LIN {X 0,Y 185.969,Z 314.942,A -85,B 0,C 180,E1 -22131.302,E2 -22131.302} C_VEL
LIN {X 0,Y 186.152,Z 314.876,A -85,B 0,C 180,E1 -22137.833,E2 -22137.833} C_VEL
LIN {X 0,Y 186.371,Z 314.881,A -85,B 0,C 180,E1 -22139.996,E2 -22139.996} C_VEL
LIN {X 0,Y 185.873,Z 314.921,A -85,B 0,C 180,E1 -22144.333,E2 -22144.333} C_VEL
LIN {X 0,Y 185.96,Z 314.906,A -85,B 0,C 180,E1 -22148.691,E2 -22148.691} C_VEL
LIN {X 0,Y 185.713,Z 314.968,A -85,B 0,C 180,E1 -22153.12,E2 -22153.12} C_VEL
LIN {X 0,Y 185.648,Z 314.931,A -85,B 0,C 180,E1 -22157.625,E2 -22157.625} C_VEL
LIN {X 0,Y 185.544,Z 314.997,A -85,B 0,C 180,E1 -22162.254,E2 -22162.254} C_VEL
LIN {X 0,Y 185.482,Z 314.953,A -85,B 0,C 180,E1 -22167.04,E2 -22167.04} C_VEL
LIN {X 0,Y 185.522,Z 315.001,A -85,B 0,C 180,E1 -22172.024,E2 -22172.024} C_VEL
LIN {X 0,Y 185.491,Z 314.96,A -85,B 0,C 180,E1 -22177.311,E2 -22177.311} C_VEL
LIN {X 0,Y 185.452,Z 315.01,A -85,B 0,C 180,E1 -22180.718,E2 -22180.718} C_VEL
LIN {X 0,Y 185.446,Z 314.975,A -85,B 0,C 180,E1 -22186.053,E2 -22186.053} C_VEL
LIN {X 0,Y 185.455,Z 315.011,A -85,B 0,C 180,E1 -22189.892,E2 -22189.892} C_VEL
LIN {X 0,Y 185.509,Z 315.032,A -85,B 0,C 180,E1 -22194.939,E2 -22194.939} C_VEL
LIN {X 0,Y 186.259,Z 317.419,A -85,B 0,C 180,E1 -22195.462,E2 -22195.462} C_VEL
LIN {X 0,Y 188.139,Z 319.677,A -85,B 0,C 180,E1 -22196.456,E2 -22196.456} C_VEL
LIN {X 0,Y 189.457,Z 320.605,A -85,B 0,C 180,E1 -22197.082,E2 -22197.082} C_VEL
LIN {X 0,Y 191.419,Z 323.893,A -85,B 0,C 180,E1 -22198.11,E2 -22198.11} C_VEL
LIN {X 0,Y 193.286,Z 325.807,A -85,B 0,C 180,E1 -22198.984,E2 -22198.984} C_VEL
LIN {X 0,Y 195.811,Z 329.375,A -85,B 0,C 180,E1 -22200.184,E2 -22200.184} C_VEL
LIN {X 0,Y 197.081,Z 331.066,A -85,B 0,C 180,E1 -22200.76,E2 -22200.76} C_VEL
LIN {X 0,Y 203.014,Z 339.247,A -85,B 0,C 180,E1 -22203.293,E2 -22203.293} C_VEL
LIN {X 0,Y 211.718,Z 352.303,A -85,B 0,C 180,E1 -22206.675,E2 -22206.675} C_VEL
LIN {X 0,Y 219.05,Z 364.426,A -85,B 0,C 180,E1 -22209.272,E2 -22209.272} C_VEL
LIN {X 0,Y 227.054,Z 378.808,A -85,B 0,C 180,E1 -22211.875,E2 -22211.875} C_VEL
LIN {X 0,Y 229.793,Z 385.325,A -85,B 0,C 180,E1 -22212.786,E2 -22212.786} C_VEL
LIN {X 0,Y 224.005,Z 468.269,A -85,B 0,C 180,E1 -22215.304,E2 -22215.304} C_VEL
LIN {X 0,Y 222.037,Z 484.164,A -85,B 0,C 180,E1 -22216.092,E2 -22216.092} C_VEL
LIN {X 0,Y 219.583,Z 498.974,A -85,B 0,C 180,E1 -22217.171,E2 -22217.171} C_VEL
LIN {X 0,Y 216.53,Z 513.139,A -85,B 0,C 180,E1 -22218.533,E2 -22218.533} C_VEL
LIN {X 0,Y 213.108,Z 526.59,A -85,B 0,C 180,E1 -22220.206,E2 -22220.206} C_VEL
LIN {X 0,Y 209.135,Z 539.856,A -85,B 0,C 180,E1 -22222.274,E2 -22222.274} C_VEL
LIN {X 0,Y 204.964,Z 552.181,A -85,B 0,C 180,E1 -22224.68,E2 -22224.68} C_VEL
LIN {X 0,Y 200.711,Z 563.728,A -85,B 0,C 180,E1 -22227.491,E2 -22227.491} C_VEL
LIN {X 0,Y 196.778,Z 573.885,A -85,B 0,C 180,E1 -22230.568,E2 -22230.568} C_VEL
LIN {X 0,Y 192.849,Z 583.499,A -85,B 0,C 180,E1 -22234.179,E2 -22234.179} C_VEL
LIN {X 0,Y 189.543,Z 591.563,A -85,B 0,C 180,E1 -22237.992,E2 -22237.992} C_VEL
LIN {X 0,Y 186.875,Z 598.44,A -85,B 0,C 180,E1 -22242.115,E2 -22242.115} C_VEL
LIN {X 0,Y 184.929,Z 604.134,A -85,B 0,C 180,E1 -22246.559,E2 -22246.559} C_VEL
LIN {X 0,Y 183.833,Z 607.594,A -85,B 0,C 180,E1 -22250.124,E2 -22250.124} C_VEL
LIN {X 0,Y 183.14,Z 609.731,A -85,B 0,C 180,E1 -22252.939,E2 -22252.939} C_VEL
LIN {X 0,Y 182.593,Z 612.209,A -85,B 0,C 180,E1 -22257.725,E2 -22257.725} C_VEL
LIN {X 0,Y 182.636,Z 613.322,A -85,B 0,C 180,E1 -22262.595,E2 -22262.595} C_VEL
LIN {X 0,Y 183.097,Z 613.279,A -85,B 0,C 180,E1 -22266.295,E2 -22266.295} C_VEL
LIN {X 0,Y 184.09,Z 612.207,A -85,B 0,C 180,E1 -22270.465,E2 -22270.465} C_VEL
LIN {X 0,Y 185.447,Z 610.546,A -85,B 0,C 180,E1 -22273.947,E2 -22273.947} C_VEL
LIN {X 0,Y 187.89,Z 607.254,A -85,B 0,C 180,E1 -22278.423,E2 -22278.423} C_VEL
LIN {X 0,Y 190.855,Z 603.121,A -85,B 0,C 180,E1 -22282.343,E2 -22282.343} C_VEL
LIN {X 0,Y 195.336,Z 596.767,A -85,B 0,C 180,E1 -22286.819,E2 -22286.819} C_VEL
LIN {X 0,Y 200.792,Z 588.688,A -85,B 0,C 180,E1 -22291.045,E2 -22291.045} C_VEL
LIN {X 0,Y 206.353,Z 580.032,A -85,B 0,C 180,E1 -22294.488,E2 -22294.488} C_VEL
LIN {X 0,Y 211.756,Z 570.942,A -85,B 0,C 180,E1 -22297.349,E2 -22297.349} C_VEL
LIN {X 0,Y 217.718,Z 560.022,A -85,B 0,C 180,E1 -22300.073,E2 -22300.073} C_VEL
LIN {X 0,Y 223.783,Z 547.561,A -85,B 0,C 180,E1 -22302.536,E2 -22302.536} C_VEL
LIN {X 0,Y 229.323,Z 534.602,A -85,B 0,C 180,E1 -22304.538,E2 -22304.538} C_VEL
LIN {X 0,Y 234.001,Z 521.869,A -85,B 0,C 180,E1 -22306.101,E2 -22306.101} C_VEL
LIN {X 0,Y 238.248,Z 507.978,A -85,B 0,C 180,E1 -22307.443,E2 -22307.443} C_VEL
LIN {X 0,Y 241.757,Z 493.694,A -85,B 0,C 180,E1 -22308.498,E2 -22308.498} C_VEL
LIN {X 0,Y 244.702,Z 478.011,A -85,B 0,C 180,E1 -22309.327,E2 -22309.327} C_VEL
LIN {X 0,Y 246.667,Z 461.81,A -85,B 0,C 180,E1 -22309.898,E2 -22309.898} C_VEL
LIN {X 0,Y 252.263,Z 398.759,A -85,B 0,C 180,E1 -22311.644,E2 -22311.644} C_VEL
LIN {X 0,Y 250.263,Z 393.549,A -85,B 0,C 180,E1 -22312.821,E2 -22312.821} C_VEL
LIN {X 0,Y 246.472,Z 386.354,A -85,B 0,C 180,E1 -22315.096,E2 -22315.096} C_VEL
LIN {X 0,Y 242.393,Z 379.192,A -85,B 0,C 180,E1 -22317.911,E2 -22317.911} C_VEL
LIN {X 0,Y 240.443,Z 376.102,A -85,B 0,C 180,E1 -22319.444,E2 -22319.444} C_VEL
LIN {X 0,Y 237.536,Z 371.34,A -85,B 0,C 180,E1 -22322.141,E2 -22322.141} C_VEL
LIN {X 0,Y 235.778,Z 368.411,A -85,B 0,C 180,E1 -22324.111,E2 -22324.111} C_VEL
LIN {X 0,Y 233.394,Z 365.664,A -85,B 0,C 180,E1 -22327.468,E2 -22327.468} C_VEL
LIN {X 0,Y 232.588,Z 363.6,A -85,B 0,C 180,E1 -22329.388,E2 -22329.388} C_VEL
LIN {X 0,Y 231.393,Z 363.089,A -85,B 0,C 180,E1 -22335.867,E2 -22335.867} C_VEL
LIN {X 0,Y 232.583,Z 363.999,A -85,B 0,C 180,E1 -22340.339,E2 -22340.339} C_VEL
LIN {X 0,Y 234.637,Z 367.807,A -85,B 0,C 180,E1 -22344.159,E2 -22344.159} C_VEL
LIN {X 0,Y 236.244,Z 370.311,A -85,B 0,C 180,E1 -22346.214,E2 -22346.214} C_VEL
LIN {X 0,Y 239.041,Z 375.498,A -85,B 0,C 180,E1 -22349.15,E2 -22349.15} C_VEL
LIN {X 0,Y 241.266,Z 379.857,A -85,B 0,C 180,E1 -22351.073,E2 -22351.073} C_VEL
LIN {X 0,Y 244.66,Z 386.769,A -85,B 0,C 180,E1 -22353.626,E2 -22353.626} C_VEL
LIN {X 0,Y 245.434,Z 389.581,A -85,B 0,C 180,E1 -22354.248,E2 -22354.248} C_VEL
LIN {X 0,Y 246.014,Z 395.44,A -85,B 0,C 180,E1 -22354.985,E2 -22354.985} C_VEL
LIN {X 0,Y 246.682,Z 402.682,A -85,B 0,C 180,E1 -22355.839,E2 -22355.839} C_VEL
LIN {X 0,Y 247.202,Z 404.751,A -85,B 0,C 180,E1 -22356.22,E2 -22356.22} C_VEL
LIN {X 0,Y 248.199,Z 407.486,A -85,B 0,C 180,E1 -22356.843,E2 -22356.843} C_VEL
LIN {X 0,Y 241.718,Z 476.664,A -85,B 0,C 180,E1 -22358.781,E2 -22358.781} C_VEL
LIN {X 0,Y 239.106,Z 492.462,A -85,B 0,C 180,E1 -22359.425,E2 -22359.425} C_VEL
LIN {X 0,Y 235.556,Z 507.607,A -85,B 0,C 180,E1 -22360.302,E2 -22360.302} C_VEL
LIN {X 0,Y 230.993,Z 522.645,A -85,B 0,C 180,E1 -22361.48,E2 -22361.48} C_VEL
LIN {X 0,Y 226.376,Z 535.543,A -85,B 0,C 180,E1 -22362.826,E2 -22362.826} C_VEL
LIN {X 0,Y 220.654,Z 549.173,A -85,B 0,C 180,E1 -22364.649,E2 -22364.649} C_VEL
LIN {X 0,Y 214.991,Z 560.943,A -85,B 0,C 180,E1 -22366.65,E2 -22366.65} C_VEL
LIN {X 0,Y 209.039,Z 572.068,A -85,B 0,C 180,E1 -22369.037,E2 -22369.037} C_VEL
LIN {X 0,Y 203.445,Z 581.51,A -85,B 0,C 180,E1 -22371.554,E2 -22371.554} C_VEL
LIN {X 0,Y 197.508,Z 590.878,A -85,B 0,C 180,E1 -22374.676,E2 -22374.676} C_VEL
LIN {X 0,Y 193.038,Z 597.736,A -85,B 0,C 180,E1 -22377.522,E2 -22377.522} C_VEL
LIN {X 0,Y 188.313,Z 604.455,A -85,B 0,C 180,E1 -22380.978,E2 -22380.978} C_VEL
LIN {X 0,Y 183.914,Z 610.718,A -85,B 0,C 180,E1 -22385.145,E2 -22385.145} C_VEL
LIN {X 0,Y 180.456,Z 615.636,A -85,B 0,C 180,E1 -22389.483,E2 -22389.483} C_VEL
LIN {X 0,Y 178.06,Z 619.319,A -85,B 0,C 180,E1 -22393.962,E2 -22393.962} C_VEL
LIN {X 0,Y 176.576,Z 621.83,A -85,B 0,C 180,E1 -22398.522,E2 -22398.522} C_VEL
LIN {X 0,Y 175.946,Z 623.194,A -85,B 0,C 180,E1 -22403.119,E2 -22403.119} C_VEL
LIN {X 0,Y 175.957,Z 623.379,A -85,B 0,C 180,E1 -22407.712,E2 -22407.712} C_VEL
LIN {X 0,Y 176.109,Z 623.043,A -85,B 0,C 180,E1 -22410.001,E2 -22410.001} C_VEL
LIN {X 0,Y 175.952,Z 621.46,A -85,B 0,C 180,E1 -22414.583,E2 -22414.583} C_VEL
LIN {X 0,Y 176.214,Z 618.649,A -85,B 0,C 180,E1 -22419.181,E2 -22419.181} C_VEL
LIN {X 0,Y 177.095,Z 614.534,A -85,B 0,C 180,E1 -22423.776,E2 -22423.776} C_VEL
LIN {X 0,Y 178.863,Z 609.007,A -85,B 0,C 180,E1 -22428.322,E2 -22428.322} C_VEL
LIN {X 0,Y 181.558,Z 601.914,A -85,B 0,C 180,E1 -22432.774,E2 -22432.774} C_VEL
LIN {X 0,Y 184.649,Z 594.281,A -85,B 0,C 180,E1 -22436.566,E2 -22436.566} C_VEL
LIN {X 0,Y 188.581,Z 585.073,A -85,B 0,C 180,E1 -22440.207,E2 -22440.207} C_VEL
LIN {X 0,Y 192.358,Z 575.617,A -85,B 0,C 180,E1 -22443.233,E2 -22443.233} C_VEL
LIN {X 0,Y 196.738,Z 564.464,A -85,B 0,C 180,E1 -22446.116,E2 -22446.116} C_VEL
LIN {X 0,Y 201.25,Z 552.272,A -85,B 0,C 180,E1 -22448.625,E2 -22448.625} C_VEL
LIN {X 0,Y 205.144,Z 540.321,A -85,B 0,C 180,E1 -22450.611,E2 -22450.611} C_VEL
LIN {X 0,Y 208.785,Z 527.578,A -85,B 0,C 180,E1 -22452.317,E2 -22452.317} C_VEL
LIN {X 0,Y 212.174,Z 513.906,A -85,B 0,C 180,E1 -22453.745,E2 -22453.745} C_VEL
LIN {X 0,Y 215.168,Z 499.638,A -85,B 0,C 180,E1 -22454.855,E2 -22454.855} C_VEL
LIN {X 0,Y 217.464,Z 484.324,A -85,B 0,C 180,E1 -22455.729,E2 -22455.729} C_VEL
LIN {X 0,Y 219.024,Z 466.927,A -85,B 0,C 180,E1 -22456.384,E2 -22456.384} C_VEL
LIN {X 0,Y 224.02,Z 395.336,A -85,B 0,C 180,E1 -22458.576,E2 -22458.576} C_VEL
LIN {X 0,Y 218.08,Z 380.998,A -85,B 0,C 180,E1 -22460.678,E2 -22460.678} C_VEL
LIN {X 0,Y 211.283,Z 366.529,A -85,B 0,C 180,E1 -22463.217,E2 -22463.217} C_VEL
LIN {X 0,Y 204.623,Z 353.731,A -85,B 0,C 180,E1 -22465.876,E2 -22465.876} C_VEL
LIN {X 0,Y 199.25,Z 344.249,A -85,B 0,C 180,E1 -22468.184,E2 -22468.184} C_VEL
LIN {X 0,Y 192.162,Z 334.537,A -85,B 0,C 180,E1 -22471.394,E2 -22471.394} C_VEL
LIN {X 0,Y 189.576,Z 330.921,A -85,B 0,C 180,E1 -22472.689,E2 -22472.689} C_VEL
LIN {X 0,Y 186.864,Z 327.443,A -85,B 0,C 180,E1 -22474.07,E2 -22474.07} C_VEL
LIN {X 0,Y 186.034,Z 326.335,A -85,B 0,C 180,E1 -22474.513,E2 -22474.513} C_VEL
LIN {X 0,Y 183.548,Z 323.572,A -85,B 0,C 180,E1 -22475.848,E2 -22475.848} C_VEL
LIN {X 0,Y 182.267,Z 321.267,A -85,B 0,C 180,E1 -22476.639,E2 -22476.639} C_VEL
LIN {X 0,Y 179.8,Z 319.198,A -85,B 0,C 180,E1 -22478.048,E2 -22478.048} C_VEL
LIN {X 0,Y 178.699,Z 317.03,A -85,B 0,C 180,E1 -22478.814,E2 -22478.814} C_VEL
LIN {X 0,Y 178.468,Z 315.883,A -85,B 0,C 180,E1 -22479.088,E2 -22479.088} C_VEL
LIN {X 0,Y 178.608,Z 315.862,A -85,B 0,C 180,E1 -22481.648,E2 -22481.648} C_VEL
LIN {X 0,Y 178.637,Z 315.809,A -85,B 0,C 180,E1 -22486.343,E2 -22486.343} C_VEL
LIN {X 0,Y 178.901,Z 315.815,A -85,B 0,C 180,E1 -22490.956,E2 -22490.956} C_VEL
LIN {X 0,Y 178.809,Z 315.792,A -85,B 0,C 180,E1 -22495.488,E2 -22495.488} C_VEL
LIN {X 0,Y 179.337,Z 315.755,A -85,B 0,C 180,E1 -22499.996,E2 -22499.996} C_VEL
LIN {X 0,Y 178.822,Z 315.795,A -85,B 0,C 180,E1 -22504.504,E2 -22504.504} C_VEL
LIN {X 0,Y 178.893,Z 315.79,A -85,B 0,C 180,E1 -22509.037,E2 -22509.037} C_VEL
LIN {X 0,Y 178.639,Z 315.838,A -85,B 0,C 180,E1 -22513.65,E2 -22513.65} C_VEL
LIN {X 0,Y 178.551,Z 315.829,A -85,B 0,C 180,E1 -22519.149,E2 -22519.149} C_VEL
LIN {X 0,Y 178.457,Z 315.841,A -85,B 0,C 180,E1 -22525.071,E2 -22525.071} C_VEL
LIN {X 0,Y 178.442,Z 315.872,A -85,B 0,C 180,E1 -22530.793,E2 -22530.793} C_VEL
LIN {X 0,Y 178.474,Z 315.852,A -85,B 0,C 180,E1 -22534.214,E2 -22534.214} C_VEL
LIN {X 0,Y 178.378,Z 315.863,A -85,B 0,C 180,E1 -22539.073,E2 -22539.073} C_VEL
LIN {X 0,Y 178.383,Z 315.887,A -85,B 0,C 180,E1 -22542.043,E2 -22542.043} C_VEL
LIN {X 0,Y 178.381,Z 315.853,A -85,B 0,C 180,E1 -22545.162,E2 -22545.162} C_VEL
LIN {X 0,Y 178.391,Z 315.884,A -85,B 0,C 180,E1 -22548.457,E2 -22548.457} C_VEL
LIN {X 0,Y 178.427,Z 316.051,A -85,B 0,C 180,E1 -22551.495,E2 -22551.495} C_VEL
LIN {X 0,Y 179.26,Z 318.459,A -85,B 0,C 180,E1 -22552.133,E2 -22552.133} C_VEL
LIN {X 0,Y 181.378,Z 320.729,A -85,B 0,C 180,E1 -22553.398,E2 -22553.398} C_VEL
LIN {X 0,Y 182.523,Z 321.562,A -85,B 0,C 180,E1 -22554.03,E2 -22554.03} C_VEL
LIN {X 0,Y 184.397,Z 324.755,A -85,B 0,C 180,E1 -22555.164,E2 -22555.164} C_VEL
LIN {X 0,Y 186.648,Z 327.025,A -85,B 0,C 180,E1 -22556.342,E2 -22556.342} C_VEL
LIN {X 0,Y 189.277,Z 330.678,A -85,B 0,C 180,E1 -22557.712,E2 -22557.712} C_VEL
LIN {X 0,Y 190.556,Z 332.255,A -85,B 0,C 180,E1 -22558.336,E2 -22558.336} C_VEL
LIN {X 0,Y 194.712,Z 338.031,A -85,B 0,C 180,E1 -22560.336,E2 -22560.336} C_VEL
LIN {X 0,Y 199.594,Z 344.846,A -85,B 0,C 180,E1 -22562.492,E2 -22562.492} C_VEL
LIN {X 0,Y 207.433,Z 356.74,A -85,B 0,C 180,E1 -22565.674,E2 -22565.674} C_VEL
LIN {X 0,Y 214.405,Z 368.342,A -85,B 0,C 180,E1 -22568.253,E2 -22568.253} C_VEL
LIN {X 0,Y 222.471,Z 383.07,A -85,B 0,C 180,E1 -22571.011,E2 -22571.011} C_VEL
LIN {X 0,Y 224.336,Z 387.564,A -85,B 0,C 180,E1 -22571.654,E2 -22571.654} C_VEL
LIN {X 0,Y 218.461,Z 468.888,A -85,B 0,C 180,E1 -22574.166,E2 -22574.166} C_VEL
LIN {X 0,Y 216.47,Z 484.361,A -85,B 0,C 180,E1 -22574.945,E2 -22574.945} C_VEL
LIN {X 0,Y 213.834,Z 499.73,A -85,B 0,C 180,E1 -22576.093,E2 -22576.093} C_VEL
LIN {X 0,Y 211.126,Z 511.825,A -85,B 0,C 180,E1 -22577.259,E2 -22577.259} C_VEL
LIN {X 0,Y 207.236,Z 526.822,A -85,B 0,C 180,E1 -22579.128,E2 -22579.128} C_VEL
LIN {X 0,Y 203.009,Z 540.396,A -85,B 0,C 180,E1 -22581.288,E2 -22581.288} C_VEL
LIN {X 0,Y 198.447,Z 553.329,A -85,B 0,C 180,E1 -22583.9,E2 -22583.9} C_VEL
LIN {X 0,Y 193.911,Z 565.051,A -85,B 0,C 180,E1 -22586.883,E2 -22586.883} C_VEL
LIN {X 0,Y 189.741,Z 575.331,A -85,B 0,C 180,E1 -22590.159,E2 -22590.159} C_VEL
LIN {X 0,Y 185.825,Z 584.495,A -85,B 0,C 180,E1 -22593.794,E2 -22593.794} C_VEL
LIN {X 0,Y 182.463,Z 592.427,A -85,B 0,C 180,E1 -22597.747,E2 -22597.747} C_VEL
LIN {X 0,Y 179.701,Z 599.325,A -85,B 0,C 180,E1 -22602.136,E2 -22602.136} C_VEL
LIN {X 0,Y 177.99,Z 604.089,A -85,B 0,C 180,E1 -22606.044,E2 -22606.044} C_VEL
LIN {X 0,Y 176.833,Z 607.616,A -85,B 0,C 180,E1 -22609.743,E2 -22609.743} C_VEL
LIN {X 0,Y 175.927,Z 610.358,A -85,B 0,C 180,E1 -22613.544,E2 -22613.544} C_VEL
LIN {X 0,Y 175.474,Z 612.543,A -85,B 0,C 180,E1 -22618.23,E2 -22618.23} C_VEL
LIN {X 0,Y 175.548,Z 613.516,A -85,B 0,C 180,E1 -22622.792,E2 -22622.792} C_VEL
LIN {X 0,Y 176.116,Z 613.448,A -85,B 0,C 180,E1 -22627.058,E2 -22627.058} C_VEL
LIN {X 0,Y 177.599,Z 611.991,A -85,B 0,C 180,E1 -22632.276,E2 -22632.276} C_VEL
LIN {X 0,Y 178.81,Z 610.595,A -85,B 0,C 180,E1 -22635.027,E2 -22635.027} C_VEL
LIN {X 0,Y 180.831,Z 608.066,A -85,B 0,C 180,E1 -22638.652,E2 -22638.652} C_VEL
LIN {X 0,Y 184.315,Z 603.615,A -85,B 0,C 180,E1 -22643.197,E2 -22643.197} C_VEL
LIN {X 0,Y 188.248,Z 598.396,A -85,B 0,C 180,E1 -22647.137,E2 -22647.137} C_VEL
LIN {X 0,Y 193.013,Z 591.885,A -85,B 0,C 180,E1 -22650.91,E2 -22650.91} C_VEL
LIN {X 0,Y 198.528,Z 583.958,A -85,B 0,C 180,E1 -22654.46,E2 -22654.46} C_VEL
LIN {X 0,Y 204.857,Z 574.171,A -85,B 0,C 180,E1 -22657.857,E2 -22657.857} C_VEL
LIN {X 0,Y 211.014,Z 563.701,A -85,B 0,C 180,E1 -22660.709,E2 -22660.709} C_VEL
LIN {X 0,Y 216.818,Z 552.838,A -85,B 0,C 180,E1 -22663.042,E2 -22663.042} C_VEL
LIN {X 0,Y 222.305,Z 541.16,A -85,B 0,C 180,E1 -22665.069,E2 -22665.069} C_VEL
LIN {X 0,Y 227.416,Z 528.817,A -85,B 0,C 180,E1 -22666.763,E2 -22666.763} C_VEL
LIN {X 0,Y 232.428,Z 514.442,A -85,B 0,C 180,E1 -22668.321,E2 -22668.321} C_VEL
LIN {X 0,Y 236.635,Z 499.469,A -85,B 0,C 180,E1 -22669.56,E2 -22669.56} C_VEL
LIN {X 0,Y 239.91,Z 484.566,A -85,B 0,C 180,E1 -22670.456,E2 -22670.456} C_VEL
LIN {X 0,Y 242.243,Z 469.817,A -85,B 0,C 180,E1 -22671.075,E2 -22671.075} C_VEL
LIN {X 0,Y 248.591,Z 401.712,A -85,B 0,C 180,E1 -22672.994,E2 -22672.994} C_VEL
LIN {X 0,Y 246.4,Z 396.681,A -85,B 0,C 180,E1 -22674.353,E2 -22674.353} C_VEL
LIN {X 0,Y 242.54,Z 389.311,A -85,B 0,C 180,E1 -22676.931,E2 -22676.931} C_VEL
LIN {X 0,Y 239.177,Z 383.222,A -85,B 0,C 180,E1 -22679.593,E2 -22679.593} C_VEL
LIN {X 0,Y 235.727,Z 377.515,A -85,B 0,C 180,E1 -22682.939,E2 -22682.939} C_VEL
LIN {X 0,Y 234.369,Z 375.198,A -85,B 0,C 180,E1 -22684.587,E2 -22684.587} C_VEL
LIN {X 0,Y 232.11,Z 372.295,A -85,B 0,C 180,E1 -22688.027,E2 -22688.027} C_VEL
LIN {X 0,Y 231.583,Z 370.675,A -85,B 0,C 180,E1 -22689.429,E2 -22689.429} C_VEL
LIN {X 0,Y 230.386,Z 370.078,A -85,B 0,C 180,E1 -22694.128,E2 -22694.128} C_VEL
LIN {X 0,Y 231.402,Z 370.743,A -85,B 0,C 180,E1 -22699.828,E2 -22699.828} C_VEL
LIN {X 0,Y 233.506,Z 374.763,A -85,B 0,C 180,E1 -22703.983,E2 -22703.983} C_VEL
LIN {X 0,Y 234.772,Z 377.041,A -85,B 0,C 180,E1 -22705.732,E2 -22705.732} C_VEL
LIN {X 0,Y 237.352,Z 381.993,A -85,B 0,C 180,E1 -22708.58,E2 -22708.58} C_VEL
LIN {X 0,Y 239.344,Z 386.127,A -85,B 0,C 180,E1 -22710.424,E2 -22710.424} C_VEL
LIN {X 0,Y 242.617,Z 393.253,A -85,B 0,C 180,E1 -22713.054,E2 -22713.054} C_VEL
LIN {X 0,Y 246.079,Z 401.676,A -85,B 0,C 180,E1 -22715.481,E2 -22715.481} C_VEL
LIN {X 0,Y 247.202,Z 404.751,A -85,B 0,C 180,E1 -22716.22,E2 -22716.22} C_VEL
LIN {X 0,Y 247.478,Z 407.165,A -85,B 0,C 180,E1 -22716.506,E2 -22716.506} C_VEL
LIN {X 0,Y 247.073,Z 410.629,A -85,B 0,C 180,E1 -22716.562,E2 -22716.562} C_VEL
LIN {X 0,Y 246.116,Z 414.43,A -85,B 0,C 180,E1 -22716.399,E2 -22716.399} C_VEL
LIN {X 0,Y 244.032,Z 421.322,A -85,B 0,C 180,E1 -22715.939,E2 -22715.939} C_VEL
LIN {X 0,Y 243.236,Z 425.628,A -85,B 0,C 180,E1 -22715.88,E2 -22715.88} C_VEL
LIN {X 0,Y 238.248,Z 476.462,A -85,B 0,C 180,E1 -22717.296,E2 -22717.296} C_VEL
LIN {X 0,Y 235.565,Z 492.245,A -85,B 0,C 180,E1 -22717.933,E2 -22717.933} C_VEL
LIN {X 0,Y 231.754,Z 507.931,A -85,B 0,C 180,E1 -22718.835,E2 -22718.835} C_VEL
LIN {X 0,Y 227.06,Z 522.856,A -85,B 0,C 180,E1 -22720.001,E2 -22720.001} C_VEL
LIN {X 0,Y 221.7,Z 537.042,A -85,B 0,C 180,E1 -22721.505,E2 -22721.505} C_VEL
LIN {X 0,Y 215.917,Z 550.055,A -85,B 0,C 180,E1 -22723.286,E2 -22723.286} C_VEL
LIN {X 0,Y 209.93,Z 561.87,A -85,B 0,C 180,E1 -22725.331,E2 -22725.331} C_VEL
LIN {X 0,Y 203.77,Z 572.85,A -85,B 0,C 180,E1 -22727.738,E2 -22727.738} C_VEL
LIN {X 0,Y 197.005,Z 583.594,A -85,B 0,C 180,E1 -22730.714,E2 -22730.714} C_VEL
LIN {X 0,Y 190.936,Z 592.566,A -85,B 0,C 180,E1 -22733.921,E2 -22733.921} C_VEL
LIN {X 0,Y 184.976,Z 601.064,A -85,B 0,C 180,E1 -22737.867,E2 -22737.867} C_VEL
LIN {X 0,Y 180.848,Z 606.356,A -85,B 0,C 180,E1 -22740.939,E2 -22740.939} C_VEL
LIN {X 0,Y 176.43,Z 612.193,A -85,B 0,C 180,E1 -22745.277,E2 -22745.277} C_VEL
LIN {X 0,Y 173.75,Z 615.698,A -85,B 0,C 180,E1 -22748.653,E2 -22748.653} C_VEL
LIN {X 0,Y 171.193,Z 619.285,A -85,B 0,C 180,E1 -22753.301,E2 -22753.301} C_VEL
LIN {X 0,Y 169.577,Z 621.717,A -85,B 0,C 180,E1 -22758.042,E2 -22758.042} C_VEL
LIN {X 0,Y 168.881,Z 623.027,A -85,B 0,C 180,E1 -22762.829,E2 -22762.829} C_VEL
LIN {X 0,Y 168.866,Z 623.155,A -85,B 0,C 180,E1 -22767.616,E2 -22767.616} C_VEL
LIN {X 0,Y 169.015,Z 622.782,A -85,B 0,C 180,E1 -22770.001,E2 -22770.001} C_VEL
LIN {X 0,Y 168.861,Z 621.126,A -85,B 0,C 180,E1 -22774.776,E2 -22774.776} C_VEL
LIN {X 0,Y 169.152,Z 618.239,A -85,B 0,C 180,E1 -22779.567,E2 -22779.567} C_VEL
LIN {X 0,Y 170.141,Z 614.043,A -85,B 0,C 180,E1 -22784.35,E2 -22784.35} C_VEL
LIN {X 0,Y 172.056,Z 608.427,A -85,B 0,C 180,E1 -22789.074,E2 -22789.074} C_VEL
LIN {X 0,Y 174.962,Z 601.239,A -85,B 0,C 180,E1 -22793.684,E2 -22793.684} C_VEL
LIN {X 0,Y 178.259,Z 593.51,A -85,B 0,C 180,E1 -22797.598,E2 -22797.598} C_VEL
LIN {X 0,Y 181.756,Z 585.608,A -85,B 0,C 180,E1 -22800.82,E2 -22800.82} C_VEL
LIN {X 0,Y 185.713,Z 576.159,A -85,B 0,C 180,E1 -22803.984,E2 -22803.984} C_VEL
LIN {X 0,Y 190.167,Z 565.306,A -85,B 0,C 180,E1 -22806.909,E2 -22806.909} C_VEL
LIN {X 0,Y 194.79,Z 553.313,A -85,B 0,C 180,E1 -22809.487,E2 -22809.487} C_VEL
LIN {X 0,Y 199.276,Z 540.18,A -85,B 0,C 180,E1 -22811.734,E2 -22811.734} C_VEL
LIN {X 0,Y 203.226,Z 526.764,A -85,B 0,C 180,E1 -22813.549,E2 -22813.549} C_VEL
LIN {X 0,Y 206.826,Z 512.678,A -85,B 0,C 180,E1 -22815.008,E2 -22815.008} C_VEL
LIN {X 0,Y 209.881,Z 498.053,A -85,B 0,C 180,E1 -22816.136,E2 -22816.136} C_VEL
LIN {X 0,Y 212.103,Z 483.191,A -85,B 0,C 180,E1 -22816.973,E2 -22816.973} C_VEL
LIN {X 0,Y 213.715,Z 465.346,A -85,B 0,C 180,E1 -22817.636,E2 -22817.636} C_VEL
LIN {X 0,Y 218.616,Z 397.485,A -85,B 0,C 180,E1 -22819.74,E2 -22819.74} C_VEL
LIN {X 0,Y 212.955,Z 383.809,A -85,B 0,C 180,E1 -22821.861,E2 -22821.861} C_VEL
LIN {X 0,Y 206.763,Z 370.469,A -85,B 0,C 180,E1 -22824.294,E2 -22824.294} C_VEL
LIN {X 0,Y 200.37,Z 357.844,A -85,B 0,C 180,E1 -22827.002,E2 -22827.002} C_VEL
LIN {X 0,Y 195.617,Z 349.465,A -85,B 0,C 180,E1 -22829.129,E2 -22829.129} C_VEL
LIN {X 0,Y 189.08,Z 340.322,A -85,B 0,C 180,E1 -22832.236,E2 -22832.236} C_VEL
LIN {X 0,Y 186.138,Z 336.31,A -85,B 0,C 180,E1 -22833.741,E2 -22833.741} C_VEL
LIN {X 0,Y 183.172,Z 332.349,A -85,B 0,C 180,E1 -22835.351,E2 -22835.351} C_VEL
LIN {X 0,Y 180.57,Z 329.169,A -85,B 0,C 180,E1 -22836.841,E2 -22836.841} C_VEL
LIN {X 0,Y 179.448,Z 327.418,A -85,B 0,C 180,E1 -22837.548,E2 -22837.548} C_VEL
LIN {X 0,Y 176.899,Z 324.763,A -85,B 0,C 180,E1 -22839.12,E2 -22839.12} C_VEL
LIN {X 0,Y 175.559,Z 322.336,A -85,B 0,C 180,E1 -22840.067,E2 -22840.067} C_VEL
LIN {X 0,Y 173.109,Z 320.353,A -85,B 0,C 180,E1 -22841.657,E2 -22841.657} C_VEL
LIN {X 0,Y 171.818,Z 318.022,A -85,B 0,C 180,E1 -22842.669,E2 -22842.669} C_VEL
LIN {X 0,Y 171.526,Z 316.748,A -85,B 0,C 180,E1 -22843.022,E2 -22843.022} C_VEL
LIN {X 0,Y 171.768,Z 316.67,A -85,B 0,C 180,E1 -22849.104,E2 -22849.104} C_VEL
LIN {X 0,Y 171.851,Z 316.699,A -85,B 0,C 180,E1 -22852.949,E2 -22852.949} C_VEL
LIN {X 0,Y 172.301,Z 316.629,A -85,B 0,C 180,E1 -22859.996,E2 -22859.996} C_VEL
LIN {X 0,Y 171.771,Z 316.669,A -85,B 0,C 180,E1 -22864.69,E2 -22864.69} C_VEL
LIN {X 0,Y 171.834,Z 316.674,A -85,B 0,C 180,E1 -22869.412,E2 -22869.412} C_VEL
LIN {X 0,Y 171.553,Z 316.707,A -85,B 0,C 180,E1 -22874.225,E2 -22874.225} C_VEL
LIN {X 0,Y 171.476,Z 316.714,A -85,B 0,C 180,E1 -22879.497,E2 -22879.497} C_VEL
LIN {X 0,Y 171.394,Z 316.714,A -85,B 0,C 180,E1 -22885.564,E2 -22885.564} C_VEL
LIN {X 0,Y 171.397,Z 316.744,A -85,B 0,C 180,E1 -22890.562,E2 -22890.562} C_VEL
LIN {X 0,Y 171.383,Z 316.723,A -85,B 0,C 180,E1 -22895.031,E2 -22895.031} C_VEL
LIN {X 0,Y 171.334,Z 316.734,A -85,B 0,C 180,E1 -22898.797,E2 -22898.797} C_VEL
LIN {X 0,Y 171.308,Z 316.737,A -85,B 0,C 180,E1 -22904.215,E2 -22904.215} C_VEL
LIN {X 0,Y 171.355,Z 316.886,A -85,B 0,C 180,E1 -22907.449,E2 -22907.449} C_VEL
LIN {X 0,Y 172.14,Z 319.223,A -85,B 0,C 180,E1 -22908.178,E2 -22908.178} C_VEL
LIN {X 0,Y 174.009,Z 321.478,A -85,B 0,C 180,E1 -22909.52,E2 -22909.52} C_VEL
LIN {X 0,Y 175.727,Z 322.713,A -85,B 0,C 180,E1 -22910.609,E2 -22910.609} C_VEL
LIN {X 0,Y 177.571,Z 325.766,A -85,B 0,C 180,E1 -22911.869,E2 -22911.869} C_VEL
LIN {X 0,Y 179.964,Z 328.066,A -85,B 0,C 180,E1 -22913.284,E2 -22913.284} C_VEL
LIN {X 0,Y 182.209,Z 331.386,A -85,B 0,C 180,E1 -22914.65,E2 -22914.65} C_VEL
LIN {X 0,Y 183.869,Z 333.183,A -85,B 0,C 180,E1 -22915.56,E2 -22915.56} C_VEL
LIN {X 0,Y 186.848,Z 337.091,A -85,B 0,C 180,E1 -22917.154,E2 -22917.154} C_VEL
LIN {X 0,Y 191.816,Z 344.118,A -85,B 0,C 180,E1 -22919.638,E2 -22919.638} C_VEL
LIN {X 0,Y 196.437,Z 350.775,A -85,B 0,C 180,E1 -22921.767,E2 -22921.767} C_VEL
LIN {X 0,Y 204.626,Z 363.438,A -85,B 0,C 180,E1 -22925.202,E2 -22925.202} C_VEL
LIN {X 0,Y 212.797,Z 377.659,A -85,B 0,C 180,E1 -22928.299,E2 -22928.299} C_VEL
LIN {X 0,Y 218.068,Z 387.703,A -85,B 0,C 180,E1 -22930.169,E2 -22930.169} C_VEL
LIN {X 0,Y 218.907,Z 389.72,A -85,B 0,C 180,E1 -22930.473,E2 -22930.473} C_VEL
LIN {X 0,Y 213.02,Z 468.937,A -85,B 0,C 180,E1 -22932.962,E2 -22932.962} C_VEL
LIN {X 0,Y 210.884,Z 484.979,A -85,B 0,C 180,E1 -22933.786,E2 -22933.786} C_VEL
LIN {X 0,Y 208.116,Z 500.331,A -85,B 0,C 180,E1 -22934.953,E2 -22934.953} C_VEL
LIN {X 0,Y 205.334,Z 512.367,A -85,B 0,C 180,E1 -22936.137,E2 -22936.137} C_VEL
LIN {X 0,Y 201.563,Z 526.45,A -85,B 0,C 180,E1 -22937.924,E2 -22937.924} C_VEL
LIN {X 0,Y 197.39,Z 539.475,A -85,B 0,C 180,E1 -22940.004,E2 -22940.004} C_VEL
LIN {X 0,Y 193.046,Z 551.515,A -85,B 0,C 180,E1 -22942.416,E2 -22942.416} C_VEL
LIN {X 0,Y 188.671,Z 562.642,A -85,B 0,C 180,E1 -22945.191,E2 -22945.191} C_VEL
LIN {X 0,Y 184.417,Z 572.84,A -85,B 0,C 180,E1 -22948.349,E2 -22948.349} C_VEL
LIN {X 0,Y 180.587,Z 581.553,A -85,B 0,C 180,E1 -22951.672,E2 -22951.672} C_VEL
LIN {X 0,Y 176.616,Z 590.378,A -85,B 0,C 180,E1 -22955.886,E2 -22955.886} C_VEL
LIN {X 0,Y 173.4,Z 597.886,A -85,B 0,C 180,E1 -22960.508,E2 -22960.508} C_VEL
LIN {X 0,Y 171.044,Z 604.02,A -85,B 0,C 180,E1 -22965.489,E2 -22965.489} C_VEL
LIN {X 0,Y 169.816,Z 607.62,A -85,B 0,C 180,E1 -22969.333,E2 -22969.333} C_VEL
LIN {X 0,Y 168.659,Z 611.144,A -85,B 0,C 180,E1 -22974.625,E2 -22974.625} C_VEL
LIN {X 0,Y 168.347,Z 612.865,A -85,B 0,C 180,E1 -22978.765,E2 -22978.765} C_VEL
LIN {X 0,Y 168.528,Z 613.751,A -85,B 0,C 180,E1 -22983.492,E2 -22983.492} C_VEL
LIN {X 0,Y 169.301,Z 613.502,A -85,B 0,C 180,E1 -22988.51,E2 -22988.51} C_VEL
LIN {X 0,Y 170.382,Z 612.579,A -85,B 0,C 180,E1 -22992.065,E2 -22992.065} C_VEL
LIN {X 0,Y 172.709,Z 610.116,A -85,B 0,C 180,E1 -22997.091,E2 -22997.091} C_VEL
LIN {X 0,Y 175.486,Z 606.888,A -85,B 0,C 180,E1 -23001.345,E2 -23001.345} C_VEL
LIN {X 0,Y 179.107,Z 602.577,A -85,B 0,C 180,E1 -23005.486,E2 -23005.486} C_VEL
LIN {X 0,Y 183.294,Z 597.357,A -85,B 0,C 180,E1 -23009.273,E2 -23009.273} C_VEL
LIN {X 0,Y 189.308,Z 589.588,A -85,B 0,C 180,E1 -23013.549,E2 -23013.549} C_VEL
LIN {X 0,Y 195.582,Z 580.874,A -85,B 0,C 180,E1 -23017.177,E2 -23017.177} C_VEL
LIN {X 0,Y 201.681,Z 571.592,A -85,B 0,C 180,E1 -23020.192,E2 -23020.192} C_VEL
LIN {X 0,Y 207.826,Z 561.379,A -85,B 0,C 180,E1 -23022.802,E2 -23022.802} C_VEL
LIN {X 0,Y 213.952,Z 549.982,A -85,B 0,C 180,E1 -23025.126,E2 -23025.126} C_VEL
LIN {X 0,Y 219.583,Z 538.113,A -85,B 0,C 180,E1 -23027.057,E2 -23027.057} C_VEL
LIN {X 0,Y 224.618,Z 525.883,A -85,B 0,C 180,E1 -23028.647,E2 -23028.647} C_VEL
LIN {X 0,Y 229.61,Z 511.42,A -85,B 0,C 180,E1 -23030.121,E2 -23030.121} C_VEL
LIN {X 0,Y 233.659,Z 496.927,A -85,B 0,C 180,E1 -23031.231,E2 -23031.231} C_VEL
LIN {X 0,Y 236.829,Z 482.241,A -85,B 0,C 180,E1 -23032.048,E2 -23032.048} C_VEL
LIN {X 0,Y 238.911,Z 468.733,A -85,B 0,C 180,E1 -23032.584,E2 -23032.584} C_VEL
LIN {X 0,Y 245.045,Z 404.917,A -85,B 0,C 180,E1 -23034.398,E2 -23034.398} C_VEL
LIN {X 0,Y 241.769,Z 398.076,A -85,B 0,C 180,E1 -23036.628,E2 -23036.628} C_VEL
LIN {X 0,Y 238.123,Z 391.047,A -85,B 0,C 180,E1 -23039.526,E2 -23039.526} C_VEL
LIN {X 0,Y 234.472,Z 384.539,A -85,B 0,C 180,E1 -23043.16,E2 -23043.16} C_VEL
LIN {X 0,Y 233.02,Z 381.981,A -85,B 0,C 180,E1 -23045.017,E2 -23045.017} C_VEL
LIN {X 0,Y 230.925,Z 379.092,A -85,B 0,C 180,E1 -23048.441,E2 -23048.441} C_VEL
LIN {X 0,Y 230.382,Z 377.624,A -85,B 0,C 180,E1 -23049.932,E2 -23049.932} C_VEL
LIN {X 0,Y 229.406,Z 377.112,A -85,B 0,C 180,E1 -23054.19,E2 -23054.19} C_VEL
LIN {X 0,Y 230.331,Z 377.763,A -85,B 0,C 180,E1 -23059.614,E2 -23059.614} C_VEL
LIN {X 0,Y 232.27,Z 381.614,A -85,B 0,C 180,E1 -23063.653,E2 -23063.653} C_VEL
LIN {X 0,Y 233.331,Z 383.672,A -85,B 0,C 180,E1 -23065.218,E2 -23065.218} C_VEL
LIN {X 0,Y 235.79,Z 388.689,A -85,B 0,C 180,E1 -23068.107,E2 -23068.107} C_VEL
LIN {X 0,Y 237.545,Z 392.682,A -85,B 0,C 180,E1 -23069.859,E2 -23069.859} C_VEL
LIN {X 0,Y 240.497,Z 399.5,A -85,B 0,C 180,E1 -23072.39,E2 -23072.39} C_VEL
LIN {X 0,Y 243.617,Z 407.584,A -85,B 0,C 180,E1 -23074.714,E2 -23074.714} C_VEL
LIN {X 0,Y 244.67,Z 410.615,A -85,B 0,C 180,E1 -23075.462,E2 -23075.462} C_VEL
LIN {X 0,Y 243.236,Z 425.628,A -85,B 0,C 180,E1 -23075.88,E2 -23075.88} C_VEL
LIN {X 0,Y 242.361,Z 431.479,A -85,B 0,C 180,E1 -23075.892,E2 -23075.892} C_VEL
LIN {X 0,Y 237.956,Z 450.603,A -85,B 0,C 180,E1 -23075.17,E2 -23075.17} C_VEL
LIN {X 0,Y 237.103,Z 456.451,A -85,B 0,C 180,E1 -23075.192,E2 -23075.192} C_VEL
LIN {X 0,Y 234.661,Z 478.558,A -85,B 0,C 180,E1 -23075.85,E2 -23075.85} C_VEL
LIN {X 0,Y 231.714,Z 494.316,A -85,B 0,C 180,E1 -23076.512,E2 -23076.512} C_VEL
LIN {X 0,Y 227.782,Z 509.385,A -85,B 0,C 180,E1 -23077.396,E2 -23077.396} C_VEL
LIN {X 0,Y 222.654,Z 524.775,A -85,B 0,C 180,E1 -23078.63,E2 -23078.63} C_VEL
LIN {X 0,Y 217.147,Z 538.563,A -85,B 0,C 180,E1 -23080.129,E2 -23080.129} C_VEL
LIN {X 0,Y 211.051,Z 551.522,A -85,B 0,C 180,E1 -23081.938,E2 -23081.938} C_VEL
LIN {X 0,Y 204.989,Z 562.853,A -85,B 0,C 180,E1 -23083.95,E2 -23083.95} C_VEL
LIN {X 0,Y 198.612,Z 573.6,A -85,B 0,C 180,E1 -23086.371,E2 -23086.371} C_VEL
LIN {X 0,Y 192.568,Z 582.77,A -85,B 0,C 180,E1 -23088.936,E2 -23088.936} C_VEL
LIN {X 0,Y 186.093,Z 591.838,A -85,B 0,C 180,E1 -23092.145,E2 -23092.145} C_VEL
LIN {X 0,Y 180.416,Z 599.424,A -85,B 0,C 180,E1 -23095.611,E2 -23095.611} C_VEL
LIN {X 0,Y 174.64,Z 606.585,A -85,B 0,C 180,E1 -23099.801,E2 -23099.801} C_VEL
LIN {X 0,Y 169.977,Z 612.308,A -85,B 0,C 180,E1 -23104.271,E2 -23104.271} C_VEL
LIN {X 0,Y 167.097,Z 615.77,A -85,B 0,C 180,E1 -23107.759,E2 -23107.759} C_VEL
LIN {X 0,Y 164.355,Z 619.267,A -85,B 0,C 180,E1 -23112.584,E2 -23112.584} C_VEL
LIN {X 0,Y 162.599,Z 621.61,A -85,B 0,C 180,E1 -23117.52,E2 -23117.52} C_VEL
LIN {X 0,Y 161.812,Z 622.84,A -85,B 0,C 180,E1 -23122.514,E2 -23122.514} C_VEL
LIN {X 0,Y 161.776,Z 622.91,A -85,B 0,C 180,E1 -23127.762,E2 -23127.762} C_VEL
LIN {X 0,Y 161.924,Z 622.521,A -85,B 0,C 180,E1 -23130.001,E2 -23130.001} C_VEL
LIN {X 0,Y 161.759,Z 620.786,A -85,B 0,C 180,E1 -23134.986,E2 -23134.986} C_VEL
LIN {X 0,Y 162.113,Z 617.817,A -85,B 0,C 180,E1 -23139.987,E2 -23139.987} C_VEL
LIN {X 0,Y 163.216,Z 613.535,A -85,B 0,C 180,E1 -23144.973,E2 -23144.973} C_VEL
LIN {X 0,Y 165.267,Z 607.824,A -85,B 0,C 180,E1 -23149.89,E2 -23149.89} C_VEL
LIN {X 0,Y 168.366,Z 600.532,A -85,B 0,C 180,E1 -23154.672,E2 -23154.672} C_VEL
LIN {X 0,Y 171.94,Z 592.699,A -85,B 0,C 180,E1 -23158.704,E2 -23158.704} C_VEL
LIN {X 0,Y 175.616,Z 584.732,A -85,B 0,C 180,E1 -23162.023,E2 -23162.023} C_VEL
LIN {X 0,Y 179.646,Z 575.445,A -85,B 0,C 180,E1 -23165.174,E2 -23165.174} C_VEL
LIN {X 0,Y 184.466,Z 564.132,A -85,B 0,C 180,E1 -23168.251,E2 -23168.251} C_VEL
LIN {X 0,Y 188.846,Z 553.136,A -85,B 0,C 180,E1 -23170.638,E2 -23170.638} C_VEL
LIN {X 0,Y 193.49,Z 540.006,A -85,B 0,C 180,E1 -23172.925,E2 -23172.925} C_VEL
LIN {X 0,Y 197.708,Z 526.156,A -85,B 0,C 180,E1 -23174.818,E2 -23174.818} C_VEL
LIN {X 0,Y 201.527,Z 511.382,A -85,B 0,C 180,E1 -23176.355,E2 -23176.355} C_VEL
LIN {X 0,Y 204.694,Z 496.405,A -85,B 0,C 180,E1 -23177.486,E2 -23177.486} C_VEL
LIN {X 0,Y 206.97,Z 480.865,A -85,B 0,C 180,E1 -23178.335,E2 -23178.335} C_VEL
LIN {X 0,Y 208.88,Z 458.536,A -85,B 0,C 180,E1 -23179.115,E2 -23179.115} C_VEL
LIN {X 0,Y 213.267,Z 399.625,A -85,B 0,C 180,E1 -23180.972,E2 -23180.972} C_VEL
LIN {X 0,Y 207.612,Z 385.876,A -85,B 0,C 180,E1 -23183.216,E2 -23183.216} C_VEL
LIN {X 0,Y 201.489,Z 372.631,A -85,B 0,C 180,E1 -23185.772,E2 -23185.772} C_VEL
LIN {X 0,Y 194.619,Z 359.167,A -85,B 0,C 180,E1 -23188.876,E2 -23188.876} C_VEL
LIN {X 0,Y 191.368,Z 353.75,A -85,B 0,C 180,E1 -23190.418,E2 -23190.418} C_VEL
LIN {X 0,Y 185.447,Z 345.265,A -85,B 0,C 180,E1 -23193.39,E2 -23193.39} C_VEL
LIN {X 0,Y 182.657,Z 341.53,A -85,B 0,C 180,E1 -23194.891,E2 -23194.891} C_VEL
LIN {X 0,Y 180.357,Z 338.323,A -85,B 0,C 180,E1 -23196.217,E2 -23196.217} C_VEL
LIN {X 0,Y 177.495,Z 334.534,A -85,B 0,C 180,E1 -23197.968,E2 -23197.968} C_VEL
LIN {X 0,Y 176.693,Z 333.457,A -85,B 0,C 180,E1 -23198.485,E2 -23198.485} C_VEL
LIN {X 0,Y 173.986,Z 330.307,A -85,B 0,C 180,E1 -23200.238,E2 -23200.238} C_VEL
LIN {X 0,Y 172.898,Z 328.58,A -85,B 0,C 180,E1 -23201.02,E2 -23201.02} C_VEL
LIN {X 0,Y 170.338,Z 325.996,A -85,B 0,C 180,E1 -23202.823,E2 -23202.823} C_VEL
LIN {X 0,Y 168.954,Z 323.332,A -85,B 0,C 180,E1 -23204,E2 -23204} C_VEL
LIN {X 0,Y 166.379,Z 321.557,A -85,B 0,C 180,E1 -23206.017,E2 -23206.017} C_VEL
LIN {X 0,Y 165.052,Z 319.377,A -85,B 0,C 180,E1 -23207.274,E2 -23207.274} C_VEL
LIN {X 0,Y 164.609,Z 317.552,A -85,B 0,C 180,E1 -23207.907,E2 -23207.907} C_VEL
LIN {X 0,Y 164.814,Z 317.578,A -85,B 0,C 180,E1 -23212.646,E2 -23212.646} C_VEL
LIN {X 0,Y 165.264,Z 317.504,A -85,B 0,C 180,E1 -23219.996,E2 -23219.996} C_VEL
LIN {X 0,Y 164.808,Z 317.525,A -85,B 0,C 180,E1 -23227.346,E2 -23227.346} C_VEL
LIN {X 0,Y 164.697,Z 317.592,A -85,B 0,C 180,E1 -23231.051,E2 -23231.051} C_VEL
LIN {X 0,Y 164.432,Z 317.57,A -85,B 0,C 180,E1 -23237.404,E2 -23237.404} C_VEL
LIN {X 0,Y 164.415,Z 317.6,A -85,B 0,C 180,E1 -23239.992,E2 -23239.992} C_VEL
LIN {X 0,Y 164.329,Z 317.588,A -85,B 0,C 180,E1 -23246.088,E2 -23246.088} C_VEL
LIN {X 0,Y 164.34,Z 317.633,A -85,B 0,C 180,E1 -23251.208,E2 -23251.208} C_VEL
LIN {X 0,Y 164.271,Z 317.599,A -85,B 0,C 180,E1 -23256.79,E2 -23256.79} C_VEL
LIN {X 0,Y 164.265,Z 317.65,A -85,B 0,C 180,E1 -23261.535,E2 -23261.535} C_VEL
LIN {X 0,Y 164.296,Z 317.748,A -85,B 0,C 180,E1 -23262.505,E2 -23262.505} C_VEL
LIN {X 0,Y 164.983,Z 319.954,A -85,B 0,C 180,E1 -23263.305,E2 -23263.305} C_VEL
LIN {X 0,Y 166.782,Z 322.217,A -85,B 0,C 180,E1 -23264.889,E2 -23264.889} C_VEL
LIN {X 0,Y 169.003,Z 323.765,A -85,B 0,C 180,E1 -23266.588,E2 -23266.588} C_VEL
LIN {X 0,Y 170.798,Z 326.879,A -85,B 0,C 180,E1 -23268.08,E2 -23268.08} C_VEL
LIN {X 0,Y 173.335,Z 329.242,A -85,B 0,C 180,E1 -23269.839,E2 -23269.839} C_VEL
LIN {X 0,Y 175.696,Z 332.6,A -85,B 0,C 180,E1 -23271.456,E2 -23271.456} C_VEL
LIN {X 0,Y 177.37,Z 334.36,A -85,B 0,C 180,E1 -23272.486,E2 -23272.486} C_VEL
LIN {X 0,Y 180.147,Z 338.071,A -85,B 0,C 180,E1 -23274.184,E2 -23274.184} C_VEL
LIN {X 0,Y 184.865,Z 344.466,A -85,B 0,C 180,E1 -23276.837,E2 -23276.837} C_VEL
LIN {X 0,Y 190.306,Z 352.086,A -85,B 0,C 180,E1 -23279.586,E2 -23279.586} C_VEL
LIN {X 0,Y 197.335,Z 362.954,A -85,B 0,C 180,E1 -23282.823,E2 -23282.823} C_VEL
LIN {X 0,Y 203.754,Z 373.563,A -85,B 0,C 180,E1 -23285.507,E2 -23285.507} C_VEL
LIN {X 0,Y 212.593,Z 389.831,A -85,B 0,C 180,E1 -23288.87,E2 -23288.87} C_VEL
LIN {X 0,Y 213.591,Z 391.977,A -85,B 0,C 180,E1 -23289.242,E2 -23289.242} C_VEL
LIN {X 0,Y 207.666,Z 469.089,A -85,B 0,C 180,E1 -23291.7,E2 -23291.7} C_VEL
LIN {X 0,Y 205.486,Z 484.989,A -85,B 0,C 180,E1 -23292.522,E2 -23292.522} C_VEL
LIN {X 0,Y 202.768,Z 499.745,A -85,B 0,C 180,E1 -23293.643,E2 -23293.643} C_VEL
LIN {X 0,Y 199.639,Z 512.897,A -85,B 0,C 180,E1 -23294.952,E2 -23294.952} C_VEL
LIN {X 0,Y 195.722,Z 526.926,A -85,B 0,C 180,E1 -23296.766,E2 -23296.766} C_VEL
LIN {X 0,Y 191.42,Z 539.894,A -85,B 0,C 180,E1 -23298.886,E2 -23298.886} C_VEL
LIN {X 0,Y 186.501,Z 552.965,A -85,B 0,C 180,E1 -23301.586,E2 -23301.586} C_VEL
LIN {X 0,Y 181.961,Z 563.956,A -85,B 0,C 180,E1 -23304.458,E2 -23304.458} C_VEL
LIN {X 0,Y 177.081,Z 575.099,A -85,B 0,C 180,E1 -23308.118,E2 -23308.118} C_VEL
LIN {X 0,Y 173.034,Z 583.852,A -85,B 0,C 180,E1 -23311.745,E2 -23311.745} C_VEL
LIN {X 0,Y 169.48,Z 591.421,A -85,B 0,C 180,E1 -23315.649,E2 -23315.649} C_VEL
LIN {X 0,Y 166.647,Z 597.729,A -85,B 0,C 180,E1 -23319.711,E2 -23319.711} C_VEL
LIN {X 0,Y 164.128,Z 603.944,A -85,B 0,C 180,E1 -23324.886,E2 -23324.886} C_VEL
LIN {X 0,Y 162.956,Z 607.248,A -85,B 0,C 180,E1 -23328.427,E2 -23328.427} C_VEL
LIN {X 0,Y 161.642,Z 611.066,A -85,B 0,C 180,E1 -23334.081,E2 -23334.081} C_VEL
LIN {X 0,Y 161.234,Z 613.188,A -85,B 0,C 180,E1 -23339.345,E2 -23339.345} C_VEL
LIN {X 0,Y 161.533,Z 614.001,A -85,B 0,C 180,E1 -23344.442,E2 -23344.442} C_VEL
LIN {X 0,Y 162.251,Z 613.786,A -85,B 0,C 180,E1 -23348.776,E2 -23348.776} C_VEL
LIN {X 0,Y 163.759,Z 612.653,A -85,B 0,C 180,E1 -23353.364,E2 -23353.364} C_VEL
LIN {X 0,Y 165.601,Z 610.844,A -85,B 0,C 180,E1 -23357.239,E2 -23357.239} C_VEL
LIN {X 0,Y 168.902,Z 607.36,A -85,B 0,C 180,E1 -23362.237,E2 -23362.237} C_VEL
LIN {X 0,Y 172.742,Z 603.141,A -85,B 0,C 180,E1 -23366.512,E2 -23366.512} C_VEL
LIN {X 0,Y 178.322,Z 596.672,A -85,B 0,C 180,E1 -23371.27,E2 -23371.27} C_VEL
LIN {X 0,Y 184.141,Z 589.541,A -85,B 0,C 180,E1 -23375.181,E2 -23375.181} C_VEL
LIN {X 0,Y 190.475,Z 581.188,A -85,B 0,C 180,E1 -23378.686,E2 -23378.686} C_VEL
LIN {X 0,Y 196.959,Z 571.809,A -85,B 0,C 180,E1 -23381.763,E2 -23381.763} C_VEL
LIN {X 0,Y 204.056,Z 560.505,A -85,B 0,C 180,E1 -23384.65,E2 -23384.65} C_VEL
LIN {X 0,Y 210.896,Z 548.133,A -85,B 0,C 180,E1 -23387.085,E2 -23387.085} C_VEL
LIN {X 0,Y 216.783,Z 535.898,A -85,B 0,C 180,E1 -23388.978,E2 -23388.978} C_VEL
LIN {X 0,Y 222.358,Z 522.322,A -85,B 0,C 180,E1 -23390.625,E2 -23390.625} C_VEL
LIN {X 0,Y 227.128,Z 508.325,A -85,B 0,C 180,E1 -23391.946,E2 -23391.946} C_VEL
LIN {X 0,Y 231.191,Z 493.334,A -85,B 0,C 180,E1 -23393.019,E2 -23393.019} C_VEL
LIN {X 0,Y 234.334,Z 477.882,A -85,B 0,C 180,E1 -23393.797,E2 -23393.797} C_VEL
LIN {X 0,Y 236.52,Z 461.332,A -85,B 0,C 180,E1 -23394.342,E2 -23394.342} C_VEL
LIN {X 0,Y 241.733,Z 408.647,A -85,B 0,C 180,E1 -23395.789,E2 -23395.789} C_VEL
LIN {X 0,Y 238.474,Z 401.722,A -85,B 0,C 180,E1 -23398.266,E2 -23398.266} C_VEL
LIN {X 0,Y 235.576,Z 396.016,A -85,B 0,C 180,E1 -23400.836,E2 -23400.836} C_VEL
LIN {X 0,Y 232.649,Z 390.601,A -85,B 0,C 180,E1 -23404.076,E2 -23404.076} C_VEL
LIN {X 0,Y 231.675,Z 388.76,A -85,B 0,C 180,E1 -23405.456,E2 -23405.456} C_VEL
LIN {X 0,Y 229.718,Z 385.804,A -85,B 0,C 180,E1 -23408.934,E2 -23408.934} C_VEL
LIN {X 0,Y 229.384,Z 384.629,A -85,B 0,C 180,E1 -23409.976,E2 -23409.976} C_VEL
LIN {X 0,Y 228.427,Z 384.121,A -85,B 0,C 180,E1 -23414.252,E2 -23414.252} C_VEL
LIN {X 0,Y 229.22,Z 384.708,A -85,B 0,C 180,E1 -23419.277,E2 -23419.277} C_VEL
LIN {X 0,Y 231.672,Z 389.617,A -85,B 0,C 180,E1 -23424.303,E2 -23424.303} C_VEL
LIN {X 0,Y 234.031,Z 394.879,A -85,B 0,C 180,E1 -23427.385,E2 -23427.385} C_VEL
LIN {X 0,Y 235.688,Z 398.982,A -85,B 0,C 180,E1 -23429.204,E2 -23429.204} C_VEL
LIN {X 0,Y 238.44,Z 405.771,A -85,B 0,C 180,E1 -23431.707,E2 -23431.707} C_VEL
LIN {X 0,Y 241.004,Z 412.828,A -85,B 0,C 180,E1 -23433.774,E2 -23433.774} C_VEL
LIN {X 0,Y 241.329,Z 413.879,A -85,B 0,C 180,E1 -23434.029,E2 -23434.029} C_VEL
LIN {X 0,Y 237.103,Z 456.451,A -85,B 0,C 180,E1 -23435.192,E2 -23435.192} C_VEL
LIN {X 0,Y 236.246,Z 462.302,A -85,B 0,C 180,E1 -23435.207,E2 -23435.207} C_VEL
LIN {X 0,Y 231.379,Z 481.332,A -85,B 0,C 180,E1 -23434.493,E2 -23434.493} C_VEL
LIN {X 0,Y 230.465,Z 485.166,A -85,B 0,C 180,E1 -23434.516,E2 -23434.516} C_VEL
LIN {X 0,Y 230.075,Z 487.078,A -85,B 0,C 180,E1 -23434.592,E2 -23434.592} C_VEL
LIN {X 0,Y 226.331,Z 503.079,A -85,B 0,C 180,E1 -23435.405,E2 -23435.405} C_VEL
LIN {X 0,Y 222.331,Z 516.128,A -85,B 0,C 180,E1 -23436.289,E2 -23436.289} C_VEL
LIN {X 0,Y 217.121,Z 530.041,A -85,B 0,C 180,E1 -23437.532,E2 -23437.532} C_VEL
LIN {X 0,Y 211.485,Z 542.816,A -85,B 0,C 180,E1 -23439.035,E2 -23439.035} C_VEL
LIN {X 0,Y 204.812,Z 555.762,A -85,B 0,C 180,E1 -23440.985,E2 -23440.985} C_VEL
LIN {X 0,Y 197.939,Z 567.59,A -85,B 0,C 180,E1 -23443.294,E2 -23443.294} C_VEL
LIN {X 0,Y 191.437,Z 577.603,A -85,B 0,C 180,E1 -23445.774,E2 -23445.774} C_VEL
LIN {X 0,Y 184.286,Z 587.45,A -85,B 0,C 180,E1 -23448.866,E2 -23448.866} C_VEL
LIN {X 0,Y 176.934,Z 596.835,A -85,B 0,C 180,E1 -23452.757,E2 -23452.757} C_VEL
LIN {X 0,Y 171.486,Z 603.505,A -85,B 0,C 180,E1 -23456.41,E2 -23456.41} C_VEL
LIN {X 0,Y 165.905,Z 609.814,A -85,B 0,C 180,E1 -23460.848,E2 -23460.848} C_VEL
LIN {X 0,Y 161.425,Z 614.771,A -85,B 0,C 180,E1 -23465.57,E2 -23465.57} C_VEL
LIN {X 0,Y 158.885,Z 617.695,A -85,B 0,C 180,E1 -23469.278,E2 -23469.278} C_VEL
LIN {X 0,Y 156.398,Z 620.52,A -85,B 0,C 180,E1 -23474.36,E2 -23474.36} C_VEL
LIN {X 0,Y 155.062,Z 622.219,A -85,B 0,C 180,E1 -23479.556,E2 -23479.556} C_VEL
LIN {X 0,Y 154.627,Z 622.814,A -85,B 0,C 180,E1 -23484.786,E2 -23484.786} C_VEL
LIN {X 0,Y 154.824,Z 622.257,A -85,B 0,C 180,E1 -23490.001,E2 -23490.001} C_VEL
LIN {X 0,Y 154.685,Z 620.447,A -85,B 0,C 180,E1 -23495.215,E2 -23495.215} C_VEL
LIN {X 0,Y 155.096,Z 617.397,A -85,B 0,C 180,E1 -23500.444,E2 -23500.444} C_VEL
LIN {X 0,Y 156.319,Z 613.028,A -85,B 0,C 180,E1 -23505.65,E2 -23505.65} C_VEL
LIN {X 0,Y 158.499,Z 607.219,A -85,B 0,C 180,E1 -23510.777,E2 -23510.777} C_VEL
LIN {X 0,Y 161.854,Z 599.829,A -85,B 0,C 180,E1 -23515.736,E2 -23515.736} C_VEL
LIN {X 0,Y 165.672,Z 591.885,A -85,B 0,C 180,E1 -23519.898,E2 -23519.898} C_VEL
LIN {X 0,Y 170.144,Z 582.403,A -85,B 0,C 180,E1 -23523.839,E2 -23523.839} C_VEL
LIN {X 0,Y 174.671,Z 572.489,A -85,B 0,C 180,E1 -23527.124,E2 -23527.124} C_VEL
LIN {X 0,Y 179.766,Z 560.847,A -85,B 0,C 180,E1 -23530.171,E2 -23530.171} C_VEL
LIN {X 0,Y 184.363,Z 549.32,A -85,B 0,C 180,E1 -23532.581,E2 -23532.581} C_VEL
LIN {X 0,Y 188.804,Z 536.943,A -85,B 0,C 180,E1 -23534.636,E2 -23534.636} C_VEL
LIN {X 0,Y 192.942,Z 523.23,A -85,B 0,C 180,E1 -23536.448,E2 -23536.448} C_VEL
LIN {X 0,Y 196.635,Z 508.96,A -85,B 0,C 180,E1 -23537.871,E2 -23537.871} C_VEL
LIN {X 0,Y 199.747,Z 493.987,A -85,B 0,C 180,E1 -23538.961,E2 -23538.961} C_VEL
LIN {X 0,Y 201.964,Z 478.535,A -85,B 0,C 180,E1 -23539.763,E2 -23539.763} C_VEL
LIN {X 0,Y 208.034,Z 401.775,A -85,B 0,C 180,E1 -23542.257,E2 -23542.257} C_VEL
LIN {X 0,Y 201.682,Z 386.459,A -85,B 0,C 180,E1 -23544.918,E2 -23544.918} C_VEL
LIN {X 0,Y 194.497,Z 371.118,A -85,B 0,C 180,E1 -23548.171,E2 -23548.171} C_VEL
LIN {X 0,Y 189.026,Z 360.621,A -85,B 0,C 180,E1 -23550.863,E2 -23550.863} C_VEL
LIN {X 0,Y 182.168,Z 350.688,A -85,B 0,C 180,E1 -23554.423,E2 -23554.423} C_VEL
LIN {X 0,Y 177.483,Z 344.181,A -85,B 0,C 180,E1 -23557.17,E2 -23557.17} C_VEL
LIN {X 0,Y 174.067,Z 339.566,A -85,B 0,C 180,E1 -23559.365,E2 -23559.365} C_VEL
LIN {X 0,Y 171.268,Z 336.042,A -85,B 0,C 180,E1 -23561.288,E2 -23561.288} C_VEL
LIN {X 0,Y 170.362,Z 334.784,A -85,B 0,C 180,E1 -23561.954,E2 -23561.954} C_VEL
LIN {X 0,Y 167.689,Z 331.654,A -85,B 0,C 180,E1 -23563.993,E2 -23563.993} C_VEL
LIN {X 0,Y 166.563,Z 329.787,A -85,B 0,C 180,E1 -23564.976,E2 -23564.976} C_VEL
LIN {X 0,Y 164.057,Z 327.615,A -85,B 0,C 180,E1 -23567.078,E2 -23567.078} C_VEL
LIN {X 0,Y 162.441,Z 324.567,A -85,B 0,C 180,E1 -23568.723,E2 -23568.723} C_VEL
LIN {X 0,Y 161.857,Z 324.05,A -85,B 0,C 180,E1 -23569.278,E2 -23569.278} C_VEL
LIN {X 0,Y 159.28,Z 322.052,A -85,B 0,C 180,E1 -23571.911,E2 -23571.911} C_VEL
LIN {X 0,Y 157.937,Z 319.577,A -85,B 0,C 180,E1 -23573.689,E2 -23573.689} C_VEL
LIN {X 0,Y 157.682,Z 318.435,A -85,B 0,C 180,E1 -23574.24,E2 -23574.24} C_VEL
LIN {X 0,Y 158.225,Z 318.378,A -85,B 0,C 180,E1 -23579.996,E2 -23579.996} C_VEL
LIN {X 0,Y 157.747,Z 318.405,A -85,B 0,C 180,E1 -23587.677,E2 -23587.677} C_VEL
LIN {X 0,Y 157.628,Z 318.474,A -85,B 0,C 180,E1 -23591.22,E2 -23591.22} C_VEL
LIN {X 0,Y 157.412,Z 318.449,A -85,B 0,C 180,E1 -23595.534,E2 -23595.534} C_VEL
LIN {X 0,Y 157.3,Z 318.504,A -85,B 0,C 180,E1 -23600.938,E2 -23600.938} C_VEL
LIN {X 0,Y 157.26,Z 318.465,A -85,B 0,C 180,E1 -23606.645,E2 -23606.645} C_VEL
LIN {X 0,Y 157.256,Z 318.521,A -85,B 0,C 180,E1 -23612.426,E2 -23612.426} C_VEL
LIN {X 0,Y 157.264,Z 318.482,A -85,B 0,C 180,E1 -23615.949,E2 -23615.949} C_VEL
LIN {X 0,Y 157.885,Z 320.73,A -85,B 0,C 180,E1 -23616.973,E2 -23616.973} C_VEL
LIN {X 0,Y 159.588,Z 322.979,A -85,B 0,C 180,E1 -23619.026,E2 -23619.026} C_VEL
LIN {X 0,Y 162.208,Z 324.709,A -85,B 0,C 180,E1 -23621.639,E2 -23621.639} C_VEL
LIN {X 0,Y 163.797,Z 327.649,A -85,B 0,C 180,E1 -23623.283,E2 -23623.283} C_VEL
LIN {X 0,Y 166.378,Z 329.822,A -85,B 0,C 180,E1 -23625.433,E2 -23625.433} C_VEL
LIN {X 0,Y 166.939,Z 330.615,A -85,B 0,C 180,E1 -23625.909,E2 -23625.909} C_VEL
LIN {X 0,Y 169.238,Z 333.94,A -85,B 0,C 180,E1 -23627.782,E2 -23627.782} C_VEL
LIN {X 0,Y 171.004,Z 335.664,A -85,B 0,C 180,E1 -23629.055,E2 -23629.055} C_VEL
LIN {X 0,Y 173.745,Z 339.338,A -85,B 0,C 180,E1 -23630.979,E2 -23630.979} C_VEL
LIN {X 0,Y 175.034,Z 340.946,A -85,B 0,C 180,E1 -23631.821,E2 -23631.821} C_VEL
LIN {X 0,Y 178.76,Z 345.902,A -85,B 0,C 180,E1 -23634.13,E2 -23634.13} C_VEL
LIN {X 0,Y 184.388,Z 353.745,A -85,B 0,C 180,E1 -23637.303,E2 -23637.303} C_VEL
LIN {X 0,Y 191.532,Z 364.572,A -85,B 0,C 180,E1 -23640.879,E2 -23640.879} C_VEL
LIN {X 0,Y 199.4,Z 377.653,A -85,B 0,C 180,E1 -23644.378,E2 -23644.378} C_VEL
LIN {X 0,Y 208.24,Z 394.242,A -85,B 0,C 180,E1 -23647.927,E2 -23647.927} C_VEL
LIN {X 0,Y 206.75,Z 415.249,A -85,B 0,C 180,E1 -23648.628,E2 -23648.628} C_VEL
LIN {X 0,Y 202.335,Z 469.666,A -85,B 0,C 180,E1 -23650.393,E2 -23650.393} C_VEL
LIN {X 0,Y 200.126,Z 485.231,A -85,B 0,C 180,E1 -23651.21,E2 -23651.21} C_VEL
LIN {X 0,Y 197.276,Z 500.238,A -85,B 0,C 180,E1 -23652.373,E2 -23652.373} C_VEL
LIN {X 0,Y 194.02,Z 513.378,A -85,B 0,C 180,E1 -23653.696,E2 -23653.696} C_VEL
LIN {X 0,Y 190.146,Z 526.834,A -85,B 0,C 180,E1 -23655.469,E2 -23655.469} C_VEL
LIN {X 0,Y 185.518,Z 540.285,A -85,B 0,C 180,E1 -23657.696,E2 -23657.696} C_VEL
LIN {X 0,Y 180.403,Z 553.382,A -85,B 0,C 180,E1 -23660.469,E2 -23660.469} C_VEL
LIN {X 0,Y 175.297,Z 565.207,A -85,B 0,C 180,E1 -23663.669,E2 -23663.669} C_VEL
LIN {X 0,Y 170.763,Z 575.122,A -85,B 0,C 180,E1 -23667.05,E2 -23667.05} C_VEL
LIN {X 0,Y 166.078,Z 584.803,A -85,B 0,C 180,E1 -23671.211,E2 -23671.211} C_VEL
LIN {X 0,Y 162.343,Z 592.43,A -85,B 0,C 180,E1 -23675.373,E2 -23675.373} C_VEL
LIN {X 0,Y 159.156,Z 599.317,A -85,B 0,C 180,E1 -23680.172,E2 -23680.172} C_VEL
LIN {X 0,Y 156.704,Z 605.229,A -85,B 0,C 180,E1 -23685.609,E2 -23685.609} C_VEL
LIN {X 0,Y 155.752,Z 607.791,A -85,B 0,C 180,E1 -23688.65,E2 -23688.65} C_VEL
LIN {X 0,Y 154.537,Z 611.284,A -85,B 0,C 180,E1 -23694.159,E2 -23694.159} C_VEL
LIN {X 0,Y 154.131,Z 613.482,A -85,B 0,C 180,E1 -23699.973,E2 -23699.973} C_VEL
LIN {X 0,Y 154.483,Z 614.217,A -85,B 0,C 180,E1 -23705.036,E2 -23705.036} C_VEL
LIN {X 0,Y 155.376,Z 613.961,A -85,B 0,C 180,E1 -23709.749,E2 -23709.749} C_VEL
LIN {X 0,Y 157.532,Z 612.369,A -85,B 0,C 180,E1 -23715.543,E2 -23715.543} C_VEL
LIN {X 0,Y 159.182,Z 610.892,A -85,B 0,C 180,E1 -23718.636,E2 -23718.636} C_VEL
LIN {X 0,Y 161.847,Z 608.362,A -85,B 0,C 180,E1 -23722.566,E2 -23722.566} C_VEL
LIN {X 0,Y 166.443,Z 603.705,A -85,B 0,C 180,E1 -23727.614,E2 -23727.614} C_VEL
LIN {X 0,Y 171.397,Z 598.343,A -85,B 0,C 180,E1 -23731.83,E2 -23731.83} C_VEL
LIN {X 0,Y 177.227,Z 591.696,A -85,B 0,C 180,E1 -23735.788,E2 -23735.788} C_VEL
LIN {X 0,Y 183.821,Z 583.693,A -85,B 0,C 180,E1 -23739.429,E2 -23739.429} C_VEL
LIN {X 0,Y 189.916,Z 575.593,A -85,B 0,C 180,E1 -23742.338,E2 -23742.338} C_VEL
LIN {X 0,Y 196.426,Z 566.151,A -85,B 0,C 180,E1 -23745.018,E2 -23745.018} C_VEL
LIN {X 0,Y 203.019,Z 555.431,A -85,B 0,C 180,E1 -23747.413,E2 -23747.413} C_VEL
LIN {X 0,Y 209.852,Z 542.776,A -85,B 0,C 180,E1 -23749.654,E2 -23749.654} C_VEL
LIN {X 0,Y 215.885,Z 529.871,A -85,B 0,C 180,E1 -23751.417,E2 -23751.417} C_VEL
LIN {X 0,Y 221.509,Z 515.462,A -85,B 0,C 180,E1 -23752.953,E2 -23752.953} C_VEL
LIN {X 0,Y 226.079,Z 500.999,A -85,B 0,C 180,E1 -23754.117,E2 -23754.117} C_VEL
LIN {X 0,Y 229.77,Z 485.846,A -85,B 0,C 180,E1 -23755.02,E2 -23755.02} C_VEL
LIN {X 0,Y 232.428,Z 470.856,A -85,B 0,C 180,E1 -23755.617,E2 -23755.617} C_VEL
LIN {X 0,Y 238.537,Z 412.454,A -85,B 0,C 180,E1 -23757.247,E2 -23757.247} C_VEL
LIN {X 0,Y 235.015,Z 404.753,A -85,B 0,C 180,E1 -23760.291,E2 -23760.291} C_VEL
LIN {X 0,Y 233.06,Z 401.075,A -85,B 0,C 180,E1 -23762.295,E2 -23762.295} C_VEL
LIN {X 0,Y 231.214,Z 397.223,A -85,B 0,C 180,E1 -23764.602,E2 -23764.602} C_VEL
LIN {X 0,Y 230.33,Z 395.536,A -85,B 0,C 180,E1 -23765.919,E2 -23765.919} C_VEL
LIN {X 0,Y 228.546,Z 392.557,A -85,B 0,C 180,E1 -23769.378,E2 -23769.378} C_VEL
LIN {X 0,Y 228.221,Z 391.578,A -85,B 0,C 180,E1 -23770.416,E2 -23770.416} C_VEL
LIN {X 0,Y 227.439,Z 391.155,A -85,B 0,C 180,E1 -23774.315,E2 -23774.315} C_VEL
LIN {X 0,Y 228.166,Z 391.729,A -85,B 0,C 180,E1 -23779.106,E2 -23779.106} C_VEL
LIN {X 0,Y 230.339,Z 396.401,A -85,B 0,C 180,E1 -23783.859,E2 -23783.859} C_VEL
LIN {X 0,Y 232.405,Z 401.381,A -85,B 0,C 180,E1 -23786.778,E2 -23786.778} C_VEL
LIN {X 0,Y 234.155,Z 405.955,A -85,B 0,C 180,E1 -23788.804,E2 -23788.804} C_VEL
LIN {X 0,Y 236.574,Z 412.359,A -85,B 0,C 180,E1 -23791.143,E2 -23791.143} C_VEL
LIN {X 0,Y 238.136,Z 417.148,A -85,B 0,C 180,E1 -23792.551,E2 -23792.551} C_VEL
LIN {X 0,Y 231.912,Z 476.496,A -85,B 0,C 180,E1 -23794.199,E2 -23794.199} C_VEL
LIN {X 0,Y 230.075,Z 487.078,A -85,B 0,C 180,E1 -23794.592,E2 -23794.592} C_VEL
LIN {X 0,Y 227.635,Z 495.599,A -85,B 0,C 180,E1 -23794.671,E2 -23794.671} C_VEL
LIN {X 0,Y 221.492,Z 510.219,A -85,B 0,C 180,E1 -23794.406,E2 -23794.406} C_VEL
LIN {X 0,Y 219.661,Z 514.767,A -85,B 0,C 180,E1 -23794.543,E2 -23794.543} C_VEL
LIN {X 0,Y 219.006,Z 516.53,A -85,B 0,C 180,E1 -23794.664,E2 -23794.664} C_VEL
LIN {X 0,Y 213.618,Z 530.403,A -85,B 0,C 180,E1 -23795.892,E2 -23795.892} C_VEL
LIN {X 0,Y 207.546,Z 543.583,A -85,B 0,C 180,E1 -23797.435,E2 -23797.435} C_VEL
LIN {X 0,Y 200.919,Z 555.918,A -85,B 0,C 180,E1 -23799.285,E2 -23799.285} C_VEL
LIN {X 0,Y 194.36,Z 566.785,A -85,B 0,C 180,E1 -23801.385,E2 -23801.385} C_VEL
LIN {X 0,Y 186.454,Z 578.337,A -85,B 0,C 180,E1 -23804.264,E2 -23804.264} C_VEL
LIN {X 0,Y 179.029,Z 588.047,A -85,B 0,C 180,E1 -23807.38,E2 -23807.38} C_VEL
LIN {X 0,Y 172.36,Z 596.146,A -85,B 0,C 180,E1 -23810.785,E2 -23810.785} C_VEL
LIN {X 0,Y 165.61,Z 603.837,A -85,B 0,C 180,E1 -23815.049,E2 -23815.049} C_VEL
LIN {X 0,Y 159.718,Z 610.017,A -85,B 0,C 180,E1 -23819.602,E2 -23819.602} C_VEL
LIN {X 0,Y 154.941,Z 614.872,A -85,B 0,C 180,E1 -23824.476,E2 -23824.476} C_VEL
LIN {X 0,Y 152.214,Z 617.743,A -85,B 0,C 180,E1 -23828.325,E2 -23828.325} C_VEL
LIN {X 0,Y 149.531,Z 620.467,A -85,B 0,C 180,E1 -23833.622,E2 -23833.622} C_VEL
LIN {X 0,Y 148.043,Z 622.076,A -85,B 0,C 180,E1 -23839.055,E2 -23839.055} C_VEL
LIN {X 0,Y 147.54,Z 622.587,A -85,B 0,C 180,E1 -23844.534,E2 -23844.534} C_VEL
LIN {X 0,Y 147.725,Z 621.972,A -85,B 0,C 180,E1 -23850.001,E2 -23850.001} C_VEL
LIN {X 0,Y 147.608,Z 620.092,A -85,B 0,C 180,E1 -23855.465,E2 -23855.465} C_VEL
LIN {X 0,Y 148.069,Z 616.953,A -85,B 0,C 180,E1 -23860.945,E2 -23860.945} C_VEL
LIN {X 0,Y 149.44,Z 612.492,A -85,B 0,C 180,E1 -23866.391,E2 -23866.391} C_VEL
LIN {X 0,Y 151.802,Z 606.58,A -85,B 0,C 180,E1 -23871.74,E2 -23871.74} C_VEL
LIN {X 0,Y 155.366,Z 599.075,A -85,B 0,C 180,E1 -23876.895,E2 -23876.895} C_VEL
LIN {X 0,Y 159.502,Z 591.016,A -85,B 0,C 180,E1 -23881.181,E2 -23881.181} C_VEL
LIN {X 0,Y 163.964,Z 581.825,A -85,B 0,C 180,E1 -23885.08,E2 -23885.08} C_VEL
LIN {X 0,Y 168.969,Z 571.303,A -85,B 0,C 180,E1 -23888.602,E2 -23888.602} C_VEL
LIN {X 0,Y 174.298,Z 559.461,A -85,B 0,C 180,E1 -23891.706,E2 -23891.706} C_VEL
LIN {X 0,Y 179.63,Z 546.388,A -85,B 0,C 180,E1 -23894.376,E2 -23894.376} C_VEL
LIN {X 0,Y 184.239,Z 533.426,A -85,B 0,C 180,E1 -23896.45,E2 -23896.45} C_VEL
LIN {X 0,Y 188.486,Z 519.269,A -85,B 0,C 180,E1 -23898.222,E2 -23898.222} C_VEL
LIN {X 0,Y 192.177,Z 504.783,A -85,B 0,C 180,E1 -23899.563,E2 -23899.563} C_VEL
LIN {X 0,Y 194.923,Z 490.919,A -85,B 0,C 180,E1 -23900.516,E2 -23900.516} C_VEL
LIN {X 0,Y 196.942,Z 476.628,A -85,B 0,C 180,E1 -23901.215,E2 -23901.215} C_VEL
LIN {X 0,Y 202.823,Z 403.905,A -85,B 0,C 180,E1 -23903.599,E2 -23903.599} C_VEL
LIN {X 0,Y 195.74,Z 386.777,A -85,B 0,C 180,E1 -23906.798,E2 -23906.798} C_VEL
LIN {X 0,Y 189.646,Z 373.9,A -85,B 0,C 180,E1 -23909.74,E2 -23909.74} C_VEL
LIN {X 0,Y 185.437,Z 365.693,A -85,B 0,C 180,E1 -23911.95,E2 -23911.95} C_VEL
LIN {X 0,Y 177.927,Z 354.428,A -85,B 0,C 180,E1 -23916.117,E2 -23916.117} C_VEL
LIN {X 0,Y 171.408,Z 345.576,A -85,B 0,C 180,E1 -23920.323,E2 -23920.323} C_VEL
LIN {X 0,Y 168.611,Z 341.811,A -85,B 0,C 180,E1 -23922.363,E2 -23922.363} C_VEL
LIN {X 0,Y 165.102,Z 337.281,A -85,B 0,C 180,E1 -23925.198,E2 -23925.198} C_VEL
LIN {X 0,Y 164.461,Z 336.289,A -85,B 0,C 180,E1 -23925.772,E2 -23925.772} C_VEL
LIN {X 0,Y 161.827,Z 333.716,A -85,B 0,C 180,E1 -23928.107,E2 -23928.107} C_VEL
LIN {X 0,Y 160.156,Z 330.783,A -85,B 0,C 180,E1 -23929.887,E2 -23929.887} C_VEL
LIN {X 0,Y 157.609,Z 328.649,A -85,B 0,C 180,E1 -23932.63,E2 -23932.63} C_VEL
LIN {X 0,Y 156.049,Z 325.673,A -85,B 0,C 180,E1 -23934.828,E2 -23934.828} C_VEL
LIN {X 0,Y 155.563,Z 325.185,A -85,B 0,C 180,E1 -23935.462,E2 -23935.462} C_VEL
LIN {X 0,Y 153.102,Z 323.474,A -85,B 0,C 180,E1 -23939.009,E2 -23939.009} C_VEL
LIN {X 0,Y 150.864,Z 320.152,A -85,B 0,C 180,E1 -23943.919,E2 -23943.919} C_VEL
LIN {X 0,Y 150.654,Z 319.294,A -85,B 0,C 180,E1 -23944.846,E2 -23944.846} C_VEL
LIN {X 0,Y 150.671,Z 319.288,A -85,B 0,C 180,E1 -23948.039,E2 -23948.039} C_VEL
LIN {X 0,Y 150.57,Z 319.354,A -85,B 0,C 180,E1 -23951.422,E2 -23951.422} C_VEL
LIN {X 0,Y 150.316,Z 319.327,A -85,B 0,C 180,E1 -23956.287,E2 -23956.287} C_VEL
LIN {X 0,Y 150.278,Z 319.371,A -85,B 0,C 180,E1 -23960.718,E2 -23960.718} C_VEL
LIN {X 0,Y 150.191,Z 319.525,A -85,B 0,C 180,E1 -23964.901,E2 -23964.901} C_VEL
LIN {X 0,Y 151.388,Z 322.564,A -85,B 0,C 180,E1 -23968.407,E2 -23968.407} C_VEL
LIN {X 0,Y 154.086,Z 324.881,A -85,B 0,C 180,E1 -23973.178,E2 -23973.178} C_VEL
LIN {X 0,Y 155.537,Z 325.578,A -85,B 0,C 180,E1 -23975.143,E2 -23975.143} C_VEL
LIN {X 0,Y 156.794,Z 328.341,A -85,B 0,C 180,E1 -23976.992,E2 -23976.992} C_VEL
LIN {X 0,Y 159.366,Z 330.698,A -85,B 0,C 180,E1 -23979.892,E2 -23979.892} C_VEL
LIN {X 0,Y 160.339,Z 331.473,A -85,B 0,C 180,E1 -23980.885,E2 -23980.885} C_VEL
LIN {X 0,Y 162.173,Z 334.493,A -85,B 0,C 180,E1 -23982.813,E2 -23982.813} C_VEL
LIN {X 0,Y 164.721,Z 336.929,A -85,B 0,C 180,E1 -23985.027,E2 -23985.027} C_VEL
LIN {X 0,Y 167.219,Z 340.463,A -85,B 0,C 180,E1 -23987.121,E2 -23987.121} C_VEL
LIN {X 0,Y 168.706,Z 342.048,A -85,B 0,C 180,E1 -23988.246,E2 -23988.246} C_VEL
LIN {X 0,Y 171.75,Z 345.978,A -85,B 0,C 180,E1 -23990.45,E2 -23990.45} C_VEL
LIN {X 0,Y 176.096,Z 352,A -85,B 0,C 180,E1 -23993.299,E2 -23993.299} C_VEL
LIN {X 0,Y 181.343,Z 359.504,A -85,B 0,C 180,E1 -23996.399,E2 -23996.399} C_VEL
LIN {X 0,Y 188.231,Z 370.181,A -85,B 0,C 180,E1 -23999.997,E2 -23999.997} C_VEL
LIN {X 0,Y 195.608,Z 382.708,A -85,B 0,C 180,E1 -24003.443,E2 -24003.443} C_VEL
LIN {X 0,Y 203.161,Z 397.129,A -85,B 0,C 180,E1 -24006.645,E2 -24006.645} C_VEL
LIN {X 0,Y 197.176,Z 469.503,A -85,B 0,C 180,E1 -24009,E2 -24009} C_VEL
LIN {X 0,Y 194.877,Z 485.334,A -85,B 0,C 180,E1 -24009.835,E2 -24009.835} C_VEL
LIN {X 0,Y 191.862,Z 500.596,A -85,B 0,C 180,E1 -24011.028,E2 -24011.028} C_VEL
LIN {X 0,Y 188.517,Z 513.7,A -85,B 0,C 180,E1 -24012.367,E2 -24012.367} C_VEL
LIN {X 0,Y 184.333,Z 527.646,A -85,B 0,C 180,E1 -24014.237,E2 -24014.237} C_VEL
LIN {X 0,Y 179.717,Z 540.565,A -85,B 0,C 180,E1 -24016.429,E2 -24016.429} C_VEL
LIN {X 0,Y 174.411,Z 553.647,A -85,B 0,C 180,E1 -24019.258,E2 -24019.258} C_VEL
LIN {X 0,Y 169.193,Z 565.235,A -85,B 0,C 180,E1 -24022.46,E2 -24022.46} C_VEL
LIN {X 0,Y 163.976,Z 576.117,A -85,B 0,C 180,E1 -24026.313,E2 -24026.313} C_VEL
LIN {X 0,Y 159.139,Z 585.652,A -85,B 0,C 180,E1 -24030.632,E2 -24030.632} C_VEL
LIN {X 0,Y 155.148,Z 593.529,A -85,B 0,C 180,E1 -24035.197,E2 -24035.197} C_VEL
LIN {X 0,Y 152.436,Z 599.113,A -85,B 0,C 180,E1 -24039.285,E2 -24039.285} C_VEL
LIN {X 0,Y 149.788,Z 605.121,A -85,B 0,C 180,E1 -24044.953,E2 -24044.953} C_VEL
LIN {X 0,Y 148.398,Z 608.601,A -85,B 0,C 180,E1 -24049.359,E2 -24049.359} C_VEL
LIN {X 0,Y 147.257,Z 612.002,A -85,B 0,C 180,E1 -24055.436,E2 -24055.436} C_VEL
LIN {X 0,Y 147.029,Z 613.752,A -85,B 0,C 180,E1 -24060.649,E2 -24060.649} C_VEL
LIN {X 0,Y 147.5,Z 614.449,A -85,B 0,C 180,E1 -24065.912,E2 -24065.912} C_VEL
LIN {X 0,Y 148.732,Z 614.043,A -85,B 0,C 180,E1 -24071.415,E2 -24071.415} C_VEL
LIN {X 0,Y 150.318,Z 613.043,A -85,B 0,C 180,E1 -24075.475,E2 -24075.475} C_VEL
LIN {X 0,Y 153.502,Z 610.452,A -85,B 0,C 180,E1 -24081.105,E2 -24081.105} C_VEL
LIN {X 0,Y 157.207,Z 607.082,A -85,B 0,C 180,E1 -24085.793,E2 -24085.793} C_VEL
LIN {X 0,Y 161.825,Z 602.629,A -85,B 0,C 180,E1 -24090.291,E2 -24090.291} C_VEL
LIN {X 0,Y 167.045,Z 597.406,A -85,B 0,C 180,E1 -24094.269,E2 -24094.269} C_VEL
LIN {X 0,Y 173.778,Z 590.086,A -85,B 0,C 180,E1 -24098.456,E2 -24098.456} C_VEL
LIN {X 0,Y 180.468,Z 582.203,A -85,B 0,C 180,E1 -24101.852,E2 -24101.852} C_VEL
LIN {X 0,Y 187.684,Z 572.808,A -85,B 0,C 180,E1 -24105.002,E2 -24105.002} C_VEL
LIN {X 0,Y 195.055,Z 562.162,A -85,B 0,C 180,E1 -24107.769,E2 -24107.769} C_VEL
LIN {X 0,Y 202.201,Z 550.464,A -85,B 0,C 180,E1 -24110.123,E2 -24110.123} C_VEL
LIN {X 0,Y 208.418,Z 538.751,A -85,B 0,C 180,E1 -24111.979,E2 -24111.979} C_VEL
LIN {X 0,Y 213.952,Z 526.734,A -85,B 0,C 180,E1 -24113.483,E2 -24113.483} C_VEL
LIN {X 0,Y 219.189,Z 513.141,A -85,B 0,C 180,E1 -24114.836,E2 -24114.836} C_VEL
LIN {X 0,Y 223.699,Z 498.825,A -85,B 0,C 180,E1 -24115.915,E2 -24115.915} C_VEL
LIN {X 0,Y 227.234,Z 484.343,A -85,B 0,C 180,E1 -24116.715,E2 -24116.715} C_VEL
LIN {X 0,Y 229.692,Z 470.537,A -85,B 0,C 180,E1 -24117.25,E2 -24117.25} C_VEL
LIN {X 0,Y 235.537,Z 416.81,A -85,B 0,C 180,E1 -24118.716,E2 -24118.716} C_VEL
LIN {X 0,Y 235.269,Z 415.841,A -85,B 0,C 180,E1 -24118.987,E2 -24118.987} C_VEL
LIN {X 0,Y 232.496,Z 409.521,A -85,B 0,C 180,E1 -24121.735,E2 -24121.735} C_VEL
LIN {X 0,Y 229.638,Z 403.466,A -85,B 0,C 180,E1 -24125.388,E2 -24125.388} C_VEL
LIN {X 0,Y 229,Z 402.323,A -85,B 0,C 180,E1 -24126.385,E2 -24126.385} C_VEL
LIN {X 0,Y 227.32,Z 399.107,A -85,B 0,C 180,E1 -24130.047,E2 -24130.047} C_VEL
LIN {X 0,Y 227.126,Z 398.577,A -85,B 0,C 180,E1 -24130.702,E2 -24130.702} C_VEL
LIN {X 0,Y 226.502,Z 398.25,A -85,B 0,C 180,E1 -24135.878,E2 -24135.878} C_VEL
LIN {X 0,Y 227.141,Z 398.917,A -85,B 0,C 180,E1 -24139.063,E2 -24139.063} C_VEL
LIN {X 0,Y 228.981,Z 403.035,A -85,B 0,C 180,E1 -24143.333,E2 -24143.333} C_VEL
LIN {X 0,Y 230.901,Z 408.075,A -85,B 0,C 180,E1 -24146.283,E2 -24146.283} C_VEL
LIN {X 0,Y 233.108,Z 414.302,A -85,B 0,C 180,E1 -24148.936,E2 -24148.936} C_VEL
LIN {X 0,Y 235.216,Z 420.655,A -85,B 0,C 180,E1 -24151.058,E2 -24151.058} C_VEL
LIN {X 0,Y 229.145,Z 476.124,A -85,B 0,C 180,E1 -24152.571,E2 -24152.571} C_VEL
LIN {X 0,Y 226.168,Z 491.862,A -85,B 0,C 180,E1 -24153.172,E2 -24153.172} C_VEL
LIN {X 0,Y 222.039,Z 507.346,A -85,B 0,C 180,E1 -24154.019,E2 -24154.019} C_VEL
LIN {X 0,Y 219.006,Z 516.53,A -85,B 0,C 180,E1 -24154.664,E2 -24154.664} C_VEL
LIN {X 0,Y 216.766,Z 521.947,A -85,B 0,C 180,E1 -24154.952,E2 -24154.952} C_VEL
LIN {X 0,Y 211.975,Z 530.572,A -85,B 0,C 180,E1 -24155.062,E2 -24155.062} C_VEL
LIN {X 0,Y 206.83,Z 538.997,A -85,B 0,C 180,E1 -24155.264,E2 -24155.264} C_VEL
LIN {X 0,Y 204.039,Z 543.9,A -85,B 0,C 180,E1 -24155.716,E2 -24155.716} C_VEL
LIN {X 0,Y 196.567,Z 557.151,A -85,B 0,C 180,E1 -24157.708,E2 -24157.708} C_VEL
LIN {X 0,Y 189.795,Z 567.786,A -85,B 0,C 180,E1 -24159.796,E2 -24159.796} C_VEL
LIN {X 0,Y 181.61,Z 579.136,A -85,B 0,C 180,E1 -24162.673,E2 -24162.673} C_VEL
LIN {X 0,Y 173.882,Z 588.638,A -85,B 0,C 180,E1 -24165.798,E2 -24165.798} C_VEL
LIN {X 0,Y 166.599,Z 596.939,A -85,B 0,C 180,E1 -24169.41,E2 -24169.41} C_VEL
LIN {X 0,Y 159.83,Z 604.181,A -85,B 0,C 180,E1 -24173.588,E2 -24173.588} C_VEL
LIN {X 0,Y 153.595,Z 610.252,A -85,B 0,C 180,E1 -24178.253,E2 -24178.253} C_VEL
LIN {X 0,Y 148.513,Z 614.977,A -85,B 0,C 180,E1 -24183.286,E2 -24183.286} C_VEL
LIN {X 0,Y 145.57,Z 617.757,A -85,B 0,C 180,E1 -24187.281,E2 -24187.281} C_VEL
LIN {X 0,Y 142.693,Z 620.424,A -85,B 0,C 180,E1 -24192.813,E2 -24192.813} C_VEL
LIN {X 0,Y 141.043,Z 621.937,A -85,B 0,C 180,E1 -24198.505,E2 -24198.505} C_VEL
LIN {X 0,Y 140.449,Z 622.359,A -85,B 0,C 180,E1 -24204.258,E2 -24204.258} C_VEL
LIN {X 0,Y 140.637,Z 621.662,A -85,B 0,C 180,E1 -24210.001,E2 -24210.001} C_VEL
LIN {X 0,Y 140.527,Z 619.734,A -85,B 0,C 180,E1 -24215.742,E2 -24215.742} C_VEL
LIN {X 0,Y 141.065,Z 616.508,A -85,B 0,C 180,E1 -24221.496,E2 -24221.496} C_VEL
LIN {X 0,Y 142.559,Z 611.948,A -85,B 0,C 180,E1 -24227.206,E2 -24227.206} C_VEL
LIN {X 0,Y 145.156,Z 605.935,A -85,B 0,C 180,E1 -24232.79,E2 -24232.79} C_VEL
LIN {X 0,Y 148.437,Z 599.35,A -85,B 0,C 180,E1 -24237.493,E2 -24237.493} C_VEL
LIN {X 0,Y 152.698,Z 591.392,A -85,B 0,C 180,E1 -24241.958,E2 -24241.958} C_VEL
LIN {X 0,Y 156.916,Z 583.293,A -85,B 0,C 180,E1 -24245.609,E2 -24245.609} C_VEL
LIN {X 0,Y 161.663,Z 573.724,A -85,B 0,C 180,E1 -24249.077,E2 -24249.077} C_VEL
LIN {X 0,Y 167.11,Z 562.394,A -85,B 0,C 180,E1 -24252.291,E2 -24252.291} C_VEL
LIN {X 0,Y 171.52,Z 552.354,A -85,B 0,C 180,E1 -24254.563,E2 -24254.563} C_VEL
LIN {X 0,Y 176.124,Z 540.611,A -85,B 0,C 180,E1 -24256.739,E2 -24256.739} C_VEL
LIN {X 0,Y 180.799,Z 527.008,A -85,B 0,C 180,E1 -24258.715,E2 -24258.715} C_VEL
LIN {X 0,Y 184.947,Z 512.652,A -85,B 0,C 180,E1 -24260.309,E2 -24260.309} C_VEL
LIN {X 0,Y 188.547,Z 497.574,A -85,B 0,C 180,E1 -24261.514,E2 -24261.514} C_VEL
LIN {X 0,Y 191.054,Z 482.885,A -85,B 0,C 180,E1 -24262.376,E2 -24262.376} C_VEL
LIN {X 0,Y 192.868,Z 465.308,A -85,B 0,C 180,E1 -24263.071,E2 -24263.071} C_VEL
LIN {X 0,Y 197.795,Z 406.289,A -85,B 0,C 180,E1 -24264.977,E2 -24264.977} C_VEL
LIN {X 0,Y 191.318,Z 390.51,A -85,B 0,C 180,E1 -24268.064,E2 -24268.064} C_VEL
LIN {X 0,Y 185.255,Z 377.225,A -85,B 0,C 180,E1 -24271.225,E2 -24271.225} C_VEL
LIN {X 0,Y 181.771,Z 370.577,A -85,B 0,C 180,E1 -24273.126,E2 -24273.126} C_VEL
LIN {X 0,Y 175.006,Z 360.198,A -85,B 0,C 180,E1 -24277.112,E2 -24277.112} C_VEL
LIN {X 0,Y 168.928,Z 351.699,A -85,B 0,C 180,E1 -24281.215,E2 -24281.215} C_VEL
LIN {X 0,Y 165.41,Z 346.986,A -85,B 0,C 180,E1 -24283.944,E2 -24283.944} C_VEL
LIN {X 0,Y 162.136,Z 342.571,A -85,B 0,C 180,E1 -24286.807,E2 -24286.807} C_VEL
LIN {X 0,Y 159.471,Z 339.532,A -85,B 0,C 180,E1 -24289.348,E2 -24289.348} C_VEL
LIN {X 0,Y 158.327,Z 337.436,A -85,B 0,C 180,E1 -24290.656,E2 -24290.656} C_VEL
LIN {X 0,Y 155.804,Z 335.064,A -85,B 0,C 180,E1 -24293.552,E2 -24293.552} C_VEL
LIN {X 0,Y 154.188,Z 332.098,A -85,B 0,C 180,E1 -24295.904,E2 -24295.904} C_VEL
LIN {X 0,Y 151.631,Z 330.097,A -85,B 0,C 180,E1 -24299.83,E2 -24299.83} C_VEL
LIN {X 0,Y 149.55,Z 326.73,A -85,B 0,C 180,E1 -24304.797,E2 -24304.797} C_VEL
LIN {X 0,Y 149.364,Z 326.28,A -85,B 0,C 180,E1 -24305.395,E2 -24305.395} C_VEL
LIN {X 0,Y 147.562,Z 325.834,A -85,B 0,C 180,E1 -24313.772,E2 -24313.772} C_VEL
LIN {X 0,Y 148.998,Z 326.456,A -85,B 0,C 180,E1 -24324.278,E2 -24324.278} C_VEL
LIN {X 0,Y 150.363,Z 329.72,A -85,B 0,C 180,E1 -24328.381,E2 -24328.381} C_VEL
LIN {X 0,Y 153.225,Z 331.998,A -85,B 0,C 180,E1 -24333.389,E2 -24333.389} C_VEL
LIN {X 0,Y 153.922,Z 332.368,A -85,B 0,C 180,E1 -24334.364,E2 -24334.364} C_VEL
LIN {X 0,Y 155.308,Z 335.183,A -85,B 0,C 180,E1 -24336.465,E2 -24336.465} C_VEL
LIN {X 0,Y 158.087,Z 337.662,A -85,B 0,C 180,E1 -24339.666,E2 -24339.666} C_VEL
LIN {X 0,Y 161.104,Z 341.887,A -85,B 0,C 180,E1 -24342.846,E2 -24342.846} C_VEL
LIN {X 0,Y 162.676,Z 343.454,A -85,B 0,C 180,E1 -24344.249,E2 -24344.249} C_VEL
LIN {X 0,Y 165.382,Z 347.153,A -85,B 0,C 180,E1 -24346.593,E2 -24346.593} C_VEL
LIN {X 0,Y 166.667,Z 348.716,A -85,B 0,C 180,E1 -24347.599,E2 -24347.599} C_VEL
LIN {X 0,Y 170.137,Z 353.479,A -85,B 0,C 180,E1 -24350.205,E2 -24350.205} C_VEL
LIN {X 0,Y 173.855,Z 358.662,A -85,B 0,C 180,E1 -24352.712,E2 -24352.712} C_VEL
LIN {X 0,Y 178.785,Z 365.967,A -85,B 0,C 180,E1 -24355.725,E2 -24355.725} C_VEL
LIN {X 0,Y 185.114,Z 376.02,A -85,B 0,C 180,E1 -24359.168,E2 -24359.168} C_VEL
LIN {X 0,Y 191.964,Z 387.994,A -85,B 0,C 180,E1 -24362.53,E2 -24362.53} C_VEL
LIN {X 0,Y 198.012,Z 399.796,A -85,B 0,C 180,E1 -24365.232,E2 -24365.232} C_VEL
LIN {X 0,Y 192.047,Z 470.068,A -85,B 0,C 180,E1 -24367.567,E2 -24367.567} C_VEL
LIN {X 0,Y 189.739,Z 485.383,A -85,B 0,C 180,E1 -24368.376,E2 -24368.376} C_VEL
LIN {X 0,Y 186.719,Z 500.281,A -85,B 0,C 180,E1 -24369.54,E2 -24369.54} C_VEL
LIN {X 0,Y 183.109,Z 514.03,A -85,B 0,C 180,E1 -24370.959,E2 -24370.959} C_VEL
LIN {X 0,Y 178.784,Z 527.946,A -85,B 0,C 180,E1 -24372.852,E2 -24372.852} C_VEL
LIN {X 0,Y 173.667,Z 541.7,A -85,B 0,C 180,E1 -24375.244,E2 -24375.244} C_VEL
LIN {X 0,Y 168.473,Z 553.925,A -85,B 0,C 180,E1 -24377.96,E2 -24377.96} C_VEL
LIN {X 0,Y 163.17,Z 565.284,A -85,B 0,C 180,E1 -24381.171,E2 -24381.171} C_VEL
LIN {X 0,Y 157.999,Z 575.638,A -85,B 0,C 180,E1 -24384.895,E2 -24384.895} C_VEL
LIN {X 0,Y 152.917,Z 585.29,A -85,B 0,C 180,E1 -24389.34,E2 -24389.34} C_VEL
LIN {X 0,Y 148.906,Z 592.755,A -85,B 0,C 180,E1 -24393.725,E2 -24393.725} C_VEL
LIN {X 0,Y 145.72,Z 598.917,A -85,B 0,C 180,E1 -24398.318,E2 -24398.318} C_VEL
LIN {X 0,Y 143.748,Z 603.078,A -85,B 0,C 180,E1 -24402.116,E2 -24402.116} C_VEL
LIN {X 0,Y 141.854,Z 607.482,A -85,B 0,C 180,E1 -24407.292,E2 -24407.292} C_VEL
LIN {X 0,Y 140.363,Z 611.341,A -85,B 0,C 180,E1 -24413.611,E2 -24413.611} C_VEL
LIN {X 0,Y 140.018,Z 612.724,A -85,B 0,C 180,E1 -24416.853,E2 -24416.853} C_VEL
LIN {X 0,Y 139.964,Z 614.021,A -85,B 0,C 180,E1 -24421.403,E2 -24421.403} C_VEL
LIN {X 0,Y 140.546,Z 614.679,A -85,B 0,C 180,E1 -24426.872,E2 -24426.872} C_VEL
LIN {X 0,Y 141.784,Z 614.32,A -85,B 0,C 180,E1 -24431.976,E2 -24431.976} C_VEL
LIN {X 0,Y 143.908,Z 613.09,A -85,B 0,C 180,E1 -24437.098,E2 -24437.098} C_VEL
LIN {X 0,Y 146.398,Z 611.236,A -85,B 0,C 180,E1 -24441.392,E2 -24441.392} C_VEL
LIN {X 0,Y 150.846,Z 607.595,A -85,B 0,C 180,E1 -24446.992,E2 -24446.992} C_VEL
LIN {X 0,Y 155.771,Z 603.274,A -85,B 0,C 180,E1 -24451.613,E2 -24451.613} C_VEL
LIN {X 0,Y 161.625,Z 597.782,A -85,B 0,C 180,E1 -24455.939,E2 -24455.939} C_VEL
LIN {X 0,Y 167.806,Z 591.466,A -85,B 0,C 180,E1 -24459.663,E2 -24459.663} C_VEL
LIN {X 0,Y 175.812,Z 582.635,A -85,B 0,C 180,E1 -24463.607,E2 -24463.607} C_VEL
LIN {X 0,Y 183.176,Z 573.549,A -85,B 0,C 180,E1 -24466.695,E2 -24466.695} C_VEL
LIN {X 0,Y 190.631,Z 563.299,A -85,B 0,C 180,E1 -24469.381,E2 -24469.381} C_VEL
LIN {X 0,Y 197.825,Z 552.097,A -85,B 0,C 180,E1 -24471.664,E2 -24471.664} C_VEL
LIN {X 0,Y 205.037,Z 539.174,A -85,B 0,C 180,E1 -24473.715,E2 -24473.715} C_VEL
LIN {X 0,Y 210.74,Z 527.285,A -85,B 0,C 180,E1 -24475.189,E2 -24475.189} C_VEL
LIN {X 0,Y 216.164,Z 513.783,A -85,B 0,C 180,E1 -24476.52,E2 -24476.52} C_VEL
LIN {X 0,Y 220.58,Z 500.382,A -85,B 0,C 180,E1 -24477.525,E2 -24477.525} C_VEL
LIN {X 0,Y 224.342,Z 485.715,A -85,B 0,C 180,E1 -24478.342,E2 -24478.342} C_VEL
LIN {X 0,Y 226.96,Z 471.787,A -85,B 0,C 180,E1 -24478.874,E2 -24478.874} C_VEL
LIN {X 0,Y 232.736,Z 420.598,A -85,B 0,C 180,E1 -24480.264,E2 -24480.264} C_VEL
LIN {X 0,Y 230.541,Z 415.3,A -85,B 0,C 180,E1 -24482.703,E2 -24482.703} C_VEL
LIN {X 0,Y 228.045,Z 409.534,A -85,B 0,C 180,E1 -24486.294,E2 -24486.294} C_VEL
LIN {X 0,Y 226.232,Z 406.086,A -85,B 0,C 180,E1 -24490.302,E2 -24490.302} C_VEL
LIN {X 0,Y 226.124,Z 405.583,A -85,B 0,C 180,E1 -24490.75,E2 -24490.75} C_VEL
LIN {X 0,Y 225.459,Z 405.216,A -85,B 0,C 180,E1 -24494.918,E2 -24494.918} C_VEL
LIN {X 0,Y 226.051,Z 405.823,A -85,B 0,C 180,E1 -24498.747,E2 -24498.747} C_VEL
LIN {X 0,Y 227.631,Z 409.716,A -85,B 0,C 180,E1 -24502.797,E2 -24502.797} C_VEL
LIN {X 0,Y 229.237,Z 414.274,A -85,B 0,C 180,E1 -24505.517,E2 -24505.517} C_VEL
LIN {X 0,Y 231.024,Z 419.666,A -85,B 0,C 180,E1 -24507.876,E2 -24507.876} C_VEL
LIN {X 0,Y 232.397,Z 424.194,A -85,B 0,C 180,E1 -24509.494,E2 -24509.494} C_VEL
LIN {X 0,Y 226.548,Z 476.137,A -85,B 0,C 180,E1 -24510.906,E2 -24510.906} C_VEL
LIN {X 0,Y 223.428,Z 492.096,A -85,B 0,C 180,E1 -24511.507,E2 -24511.507} C_VEL
LIN {X 0,Y 219.298,Z 507.143,A -85,B 0,C 180,E1 -24512.304,E2 -24512.304} C_VEL
LIN {X 0,Y 214.44,Z 521.067,A -85,B 0,C 180,E1 -24513.311,E2 -24513.311} C_VEL
LIN {X 0,Y 208.951,Z 533.92,A -85,B 0,C 180,E1 -24514.511,E2 -24514.511} C_VEL
LIN {X 0,Y 204.039,Z 543.9,A -85,B 0,C 180,E1 -24515.716,E2 -24515.716} C_VEL
LIN {X 0,Y 201.971,Z 547.248,A -85,B 0,C 180,E1 -24515.99,E2 -24515.99} C_VEL
LIN {X 0,Y 193.276,Z 557.551,A -85,B 0,C 180,E1 -24516.07,E2 -24516.07} C_VEL
LIN {X 0,Y 191.036,Z 560.576,A -85,B 0,C 180,E1 -24516.444,E2 -24516.444} C_VEL
LIN {X 0,Y 184.129,Z 570.555,A -85,B 0,C 180,E1 -24518.516,E2 -24518.516} C_VEL
LIN {X 0,Y 175.711,Z 581.407,A -85,B 0,C 180,E1 -24521.416,E2 -24521.416} C_VEL
LIN {X 0,Y 167.802,Z 590.489,A -85,B 0,C 180,E1 -24524.604,E2 -24524.604} C_VEL
LIN {X 0,Y 159.567,Z 599.106,A -85,B 0,C 180,E1 -24528.652,E2 -24528.652} C_VEL
LIN {X 0,Y 152.37,Z 606.098,A -85,B 0,C 180,E1 -24533.16,E2 -24533.16} C_VEL
LIN {X 0,Y 146.121,Z 611.711,A -85,B 0,C 180,E1 -24538.06,E2 -24538.06} C_VEL
LIN {X 0,Y 141.021,Z 616.05,A -85,B 0,C 180,E1 -24543.353,E2 -24543.353} C_VEL
LIN {X 0,Y 137.264,Z 619.212,A -85,B 0,C 180,E1 -24549,E2 -24549} C_VEL
LIN {X 0,Y 134.765,Z 621.227,A -85,B 0,C 180,E1 -24554.887,E2 -24554.887} C_VEL
LIN {X 0,Y 133.579,Z 622.102,A -85,B 0,C 180,E1 -24560.92,E2 -24560.92} C_VEL
LIN {X 0,Y 133.398,Z 621.88,A -85,B 0,C 180,E1 -24566.981,E2 -24566.981} C_VEL
LIN {X 0,Y 133.541,Z 621.343,A -85,B 0,C 180,E1 -24570.001,E2 -24570.001} C_VEL
LIN {X 0,Y 133.439,Z 619.337,A -85,B 0,C 180,E1 -24576.048,E2 -24576.048} C_VEL
LIN {X 0,Y 134.062,Z 616.052,A -85,B 0,C 180,E1 -24582.105,E2 -24582.105} C_VEL
LIN {X 0,Y 135.718,Z 611.396,A -85,B 0,C 180,E1 -24588.102,E2 -24588.102} C_VEL
LIN {X 0,Y 138.76,Z 604.913,A -85,B 0,C 180,E1 -24594.253,E2 -24594.253} C_VEL
LIN {X 0,Y 142.676,Z 597.545,A -85,B 0,C 180,E1 -24599.511,E2 -24599.511} C_VEL
LIN {X 0,Y 147.381,Z 589.238,A -85,B 0,C 180,E1 -24604.078,E2 -24604.078} C_VEL
LIN {X 0,Y 152.27,Z 579.861,A -85,B 0,C 180,E1 -24608.168,E2 -24608.168} C_VEL
LIN {X 0,Y 157.96,Z 568.899,A -85,B 0,C 180,E1 -24611.866,E2 -24611.866} C_VEL
LIN {X 0,Y 163.296,Z 557.742,A -85,B 0,C 180,E1 -24614.81,E2 -24614.81} C_VEL
LIN {X 0,Y 168.531,Z 545.705,A -85,B 0,C 180,E1 -24617.306,E2 -24617.306} C_VEL
LIN {X 0,Y 173.396,Z 532.939,A -85,B 0,C 180,E1 -24619.389,E2 -24619.389} C_VEL
LIN {X 0,Y 178.055,Z 518.459,A -85,B 0,C 180,E1 -24621.218,E2 -24621.218} C_VEL
LIN {X 0,Y 181.973,Z 503.851,A -85,B 0,C 180,E1 -24622.575,E2 -24622.575} C_VEL
LIN {X 0,Y 185.019,Z 488.885,A -85,B 0,C 180,E1 -24623.592,E2 -24623.592} C_VEL
LIN {X 0,Y 187.145,Z 473.643,A -85,B 0,C 180,E1 -24624.301,E2 -24624.301} C_VEL
LIN {X 0,Y 192.784,Z 408.556,A -85,B 0,C 180,E1 -24626.451,E2 -24626.451} C_VEL
LIN {X 0,Y 186.953,Z 394.134,A -85,B 0,C 180,E1 -24629.412,E2 -24629.412} C_VEL
LIN {X 0,Y 181.863,Z 382.708,A -85,B 0,C 180,E1 -24632.212,E2 -24632.212} C_VEL
LIN {X 0,Y 178.473,Z 375.948,A -85,B 0,C 180,E1 -24634.181,E2 -24634.181} C_VEL
LIN {X 0,Y 172.183,Z 366.024,A -85,B 0,C 180,E1 -24638.074,E2 -24638.074} C_VEL
LIN {X 0,Y 166.586,Z 357.933,A -85,B 0,C 180,E1 -24642.056,E2 -24642.056} C_VEL
LIN {X 0,Y 162.96,Z 353.005,A -85,B 0,C 180,E1 -24644.999,E2 -24644.999} C_VEL
LIN {X 0,Y 160.1,Z 349.015,A -85,B 0,C 180,E1 -24647.647,E2 -24647.647} C_VEL
LIN {X 0,Y 157.326,Z 345.541,A -85,B 0,C 180,E1 -24650.474,E2 -24650.474} C_VEL
LIN {X 0,Y 156.444,Z 344.008,A -85,B 0,C 180,E1 -24651.532,E2 -24651.532} C_VEL
LIN {X 0,Y 154.01,Z 341.403,A -85,B 0,C 180,E1 -24654.545,E2 -24654.545} C_VEL
LIN {X 0,Y 152.701,Z 338.935,A -85,B 0,C 180,E1 -24656.521,E2 -24656.521} C_VEL
LIN {X 0,Y 150.177,Z 336.685,A -85,B 0,C 180,E1 -24660.708,E2 -24660.708} C_VEL
LIN {X 0,Y 148.111,Z 333.241,A -85,B 0,C 180,E1 -24666.125,E2 -24666.125} C_VEL
LIN {X 0,Y 146.586,Z 332.863,A -85,B 0,C 180,E1 -24673.865,E2 -24673.865} C_VEL
LIN {X 0,Y 147.478,Z 333.309,A -85,B 0,C 180,E1 -24682.405,E2 -24682.405} C_VEL
LIN {X 0,Y 147.899,Z 333.617,A -85,B 0,C 180,E1 -24683.98,E2 -24683.98} C_VEL
LIN {X 0,Y 149.223,Z 336.705,A -85,B 0,C 180,E1 -24688.092,E2 -24688.092} C_VEL
LIN {X 0,Y 152.467,Z 339.444,A -85,B 0,C 180,E1 -24693.797,E2 -24693.797} C_VEL
LIN {X 0,Y 154.311,Z 342.591,A -85,B 0,C 180,E1 -24696.551,E2 -24696.551} C_VEL
LIN {X 0,Y 156.723,Z 344.822,A -85,B 0,C 180,E1 -24699.379,E2 -24699.379} C_VEL
LIN {X 0,Y 159.135,Z 348.328,A -85,B 0,C 180,E1 -24702.014,E2 -24702.014} C_VEL
LIN {X 0,Y 160.693,Z 349.996,A -85,B 0,C 180,E1 -24703.488,E2 -24703.488} C_VEL
LIN {X 0,Y 163.431,Z 353.725,A -85,B 0,C 180,E1 -24705.95,E2 -24705.95} C_VEL
LIN {X 0,Y 167.639,Z 359.558,A -85,B 0,C 180,E1 -24709.285,E2 -24709.285} C_VEL
LIN {X 0,Y 172.627,Z 366.676,A -85,B 0,C 180,E1 -24712.752,E2 -24712.752} C_VEL
LIN {X 0,Y 179.295,Z 377.295,A -85,B 0,C 180,E1 -24716.818,E2 -24716.818} C_VEL
LIN {X 0,Y 186.755,Z 390.199,A -85,B 0,C 180,E1 -24720.774,E2 -24720.774} C_VEL
LIN {X 0,Y 193.081,Z 402.588,A -85,B 0,C 180,E1 -24723.81,E2 -24723.81} C_VEL
LIN {X 0,Y 187.089,Z 469.977,A -85,B 0,C 180,E1 -24726.035,E2 -24726.035} C_VEL
LIN {X 0,Y 184.627,Z 485.862,A -85,B 0,C 180,E1 -24726.886,E2 -24726.886} C_VEL
LIN {X 0,Y 181.447,Z 500.865,A -85,B 0,C 180,E1 -24728.07,E2 -24728.07} C_VEL
LIN {X 0,Y 177.804,Z 514.253,A -85,B 0,C 180,E1 -24729.463,E2 -24729.463} C_VEL
LIN {X 0,Y 173.323,Z 528.169,A -85,B 0,C 180,E1 -24731.378,E2 -24731.378} C_VEL
LIN {X 0,Y 168.503,Z 540.759,A -85,B 0,C 180,E1 -24733.578,E2 -24733.578} C_VEL
LIN {X 0,Y 163.133,Z 553.031,A -85,B 0,C 180,E1 -24736.293,E2 -24736.293} C_VEL
LIN {X 0,Y 157.344,Z 565.043,A -85,B 0,C 180,E1 -24739.707,E2 -24739.707} C_VEL
LIN {X 0,Y 152.134,Z 575.065,A -85,B 0,C 180,E1 -24743.367,E2 -24743.367} C_VEL
LIN {X 0,Y 146.748,Z 584.873,A -85,B 0,C 180,E1 -24747.941,E2 -24747.941} C_VEL
LIN {X 0,Y 142.182,Z 592.964,A -85,B 0,C 180,E1 -24752.832,E2 -24752.832} C_VEL
LIN {X 0,Y 139.063,Z 598.691,A -85,B 0,C 180,E1 -24757.257,E2 -24757.257} C_VEL
LIN {X 0,Y 136.551,Z 603.717,A -85,B 0,C 180,E1 -24762.099,E2 -24762.099} C_VEL
LIN {X 0,Y 134.894,Z 607.395,A -85,B 0,C 180,E1 -24766.65,E2 -24766.65} C_VEL
LIN {X 0,Y 133.592,Z 610.506,A -85,B 0,C 180,E1 -24771.606,E2 -24771.606} C_VEL
LIN {X 0,Y 133.008,Z 612.529,A -85,B 0,C 180,E1 -24776.083,E2 -24776.083} C_VEL
LIN {X 0,Y 132.891,Z 614.281,A -85,B 0,C 180,E1 -24782.214,E2 -24782.214} C_VEL
LIN {X 0,Y 133.605,Z 614.9,A -85,B 0,C 180,E1 -24787.914,E2 -24787.914} C_VEL
LIN {X 0,Y 135.042,Z 614.507,A -85,B 0,C 180,E1 -24793.239,E2 -24793.239} C_VEL
LIN {X 0,Y 138.078,Z 612.813,A -85,B 0,C 180,E1 -24799.769,E2 -24799.769} C_VEL
LIN {X 0,Y 140.348,Z 611.285,A -85,B 0,C 180,E1 -24803.242,E2 -24803.242} C_VEL
LIN {X 0,Y 143.82,Z 608.74,A -85,B 0,C 180,E1 -24807.49,E2 -24807.49} C_VEL
LIN {X 0,Y 149.792,Z 603.918,A -85,B 0,C 180,E1 -24813.051,E2 -24813.051} C_VEL
LIN {X 0,Y 157.091,Z 597.491,A -85,B 0,C 180,E1 -24818.168,E2 -24818.168} C_VEL
LIN {X 0,Y 164.139,Z 590.713,A -85,B 0,C 180,E1 -24822.125,E2 -24822.125} C_VEL
LIN {X 0,Y 172.18,Z 582.183,A -85,B 0,C 180,E1 -24825.828,E2 -24825.828} C_VEL
LIN {X 0,Y 180.539,Z 572.217,A -85,B 0,C 180,E1 -24829.085,E2 -24829.085} C_VEL
LIN {X 0,Y 189.008,Z 560.795,A -85,B 0,C 180,E1 -24831.892,E2 -24831.892} C_VEL
LIN {X 0,Y 196.25,Z 549.615,A -85,B 0,C 180,E1 -24834.017,E2 -24834.017} C_VEL
LIN {X 0,Y 203.221,Z 537.205,A -85,B 0,C 180,E1 -24835.839,E2 -24835.839} C_VEL
LIN {X 0,Y 209.305,Z 524.395,A -85,B 0,C 180,E1 -24837.319,E2 -24837.319} C_VEL
LIN {X 0,Y 214.842,Z 510.352,A -85,B 0,C 180,E1 -24838.569,E2 -24838.569} C_VEL
LIN {X 0,Y 219.647,Z 495.042,A -85,B 0,C 180,E1 -24839.603,E2 -24839.603} C_VEL
LIN {X 0,Y 223.281,Z 479.527,A -85,B 0,C 180,E1 -24840.336,E2 -24840.336} C_VEL
LIN {X 0,Y 225.68,Z 464.107,A -85,B 0,C 180,E1 -24840.82,E2 -24840.82} C_VEL
LIN {X 0,Y 230.147,Z 424.843,A -85,B 0,C 180,E1 -24841.842,E2 -24841.842} C_VEL
LIN {X 0,Y 228.77,Z 421.436,A -85,B 0,C 180,E1 -24843.525,E2 -24843.525} C_VEL
LIN {X 0,Y 226.713,Z 416.222,A -85,B 0,C 180,E1 -24846.806,E2 -24846.806} C_VEL
LIN {X 0,Y 225.118,Z 412.926,A -85,B 0,C 180,E1 -24850.688,E2 -24850.688} C_VEL
LIN {X 0,Y 224.913,Z 412.489,A -85,B 0,C 180,E1 -24851.54,E2 -24851.54} C_VEL
LIN {X 0,Y 224.591,Z 412.349,A -85,B 0,C 180,E1 -24856.36,E2 -24856.36} C_VEL
LIN {X 0,Y 224.983,Z 412.856,A -85,B 0,C 180,E1 -24858.522,E2 -24858.522} C_VEL
LIN {X 0,Y 226.336,Z 416.474,A -85,B 0,C 180,E1 -24862.322,E2 -24862.322} C_VEL
LIN {X 0,Y 227.752,Z 420.778,A -85,B 0,C 180,E1 -24864.903,E2 -24864.903} C_VEL
LIN {X 0,Y 229.821,Z 427.737,A -85,B 0,C 180,E1 -24867.847,E2 -24867.847} C_VEL
LIN {X 0,Y 229.754,Z 429.181,A -85,B 0,C 180,E1 -24867.967,E2 -24867.967} C_VEL
LIN {X 0,Y 224.299,Z 475.515,A -85,B 0,C 180,E1 -24869.18,E2 -24869.18} C_VEL
LIN {X 0,Y 221.202,Z 491.157,A -85,B 0,C 180,E1 -24869.745,E2 -24869.745} C_VEL
LIN {X 0,Y 217.139,Z 505.837,A -85,B 0,C 180,E1 -24870.489,E2 -24870.489} C_VEL
LIN {X 0,Y 212.128,Z 519.979,A -85,B 0,C 180,E1 -24871.451,E2 -24871.451} C_VEL
LIN {X 0,Y 206.484,Z 532.961,A -85,B 0,C 180,E1 -24872.609,E2 -24872.609} C_VEL
LIN {X 0,Y 199.662,Z 546.309,A -85,B 0,C 180,E1 -24874.194,E2 -24874.194} C_VEL
LIN {X 0,Y 191.702,Z 559.549,A -85,B 0,C 180,E1 -24876.244,E2 -24876.244} C_VEL
LIN {X 0,Y 191.036,Z 560.576,A -85,B 0,C 180,E1 -24876.444,E2 -24876.444} C_VEL
LIN {X 0,Y 187.809,Z 564.991,A -85,B 0,C 180,E1 -24877.143,E2 -24877.143} C_VEL
LIN {X 0,Y 181.316,Z 572.063,A -85,B 0,C 180,E1 -24877.906,E2 -24877.906} C_VEL
LIN {X 0,Y 174.542,Z 578.753,A -85,B 0,C 180,E1 -24878.798,E2 -24878.798} C_VEL
LIN {X 0,Y 170.921,Z 582.482,A -85,B 0,C 180,E1 -24879.724,E2 -24879.724} C_VEL
LIN {X 0,Y 161.785,Z 592.271,A -85,B 0,C 180,E1 -24883.315,E2 -24883.315} C_VEL
LIN {X 0,Y 154.327,Z 599.595,A -85,B 0,C 180,E1 -24886.917,E2 -24886.917} C_VEL
LIN {X 0,Y 146.746,Z 606.446,A -85,B 0,C 180,E1 -24891.496,E2 -24891.496} C_VEL
LIN {X 0,Y 140.105,Z 611.908,A -85,B 0,C 180,E1 -24896.513,E2 -24896.513} C_VEL
LIN {X 0,Y 134.675,Z 616.129,A -85,B 0,C 180,E1 -24901.99,E2 -24901.99} C_VEL
LIN {X 0,Y 130.595,Z 619.185,A -85,B 0,C 180,E1 -24907.872,E2 -24907.872} C_VEL
LIN {X 0,Y 127.862,Z 621.128,A -85,B 0,C 180,E1 -24914.05,E2 -24914.05} C_VEL
LIN {X 0,Y 126.542,Z 621.92,A -85,B 0,C 180,E1 -24920.41,E2 -24920.41} C_VEL
LIN {X 0,Y 126.302,Z 621.604,A -85,B 0,C 180,E1 -24926.812,E2 -24926.812} C_VEL
LIN {X 0,Y 126.454,Z 621.021,A -85,B 0,C 180,E1 -24930.001,E2 -24930.001} C_VEL
LIN {X 0,Y 126.356,Z 618.917,A -85,B 0,C 180,E1 -24936.388,E2 -24936.388} C_VEL
LIN {X 0,Y 127.061,Z 615.543,A -85,B 0,C 180,E1 -24942.783,E2 -24942.783} C_VEL
LIN {X 0,Y 128.922,Z 610.808,A -85,B 0,C 180,E1 -24949.093,E2 -24949.093} C_VEL
LIN {X 0,Y 132.02,Z 604.579,A -85,B 0,C 180,E1 -24955.207,E2 -24955.207} C_VEL
LIN {X 0,Y 135.82,Z 597.762,A -85,B 0,C 180,E1 -24960.3,E2 -24960.3} C_VEL
LIN {X 0,Y 140.715,Z 589.549,A -85,B 0,C 180,E1 -24965.056,E2 -24965.056} C_VEL
LIN {X 0,Y 145.364,Z 581.127,A -85,B 0,C 180,E1 -24968.941,E2 -24968.941} C_VEL
LIN {X 0,Y 150.752,Z 571.254,A -85,B 0,C 180,E1 -24972.531,E2 -24972.531} C_VEL
LIN {X 0,Y 156.71,Z 559.51,A -85,B 0,C 180,E1 -24975.853,E2 -24975.853} C_VEL
LIN {X 0,Y 162.095,Z 547.879,A -85,B 0,C 180,E1 -24978.41,E2 -24978.41} C_VEL
LIN {X 0,Y 166.901,Z 536.159,A -85,B 0,C 180,E1 -24980.452,E2 -24980.452} C_VEL
LIN {X 0,Y 171.832,Z 521.836,A -85,B 0,C 180,E1 -24982.415,E2 -24982.415} C_VEL
LIN {X 0,Y 176.118,Z 506.988,A -85,B 0,C 180,E1 -24983.908,E2 -24983.908} C_VEL
LIN {X 0,Y 179.425,Z 492.423,A -85,B 0,C 180,E1 -24984.973,E2 -24984.973} C_VEL
LIN {X 0,Y 181.946,Z 476.603,A -85,B 0,C 180,E1 -24985.777,E2 -24985.777} C_VEL
LIN {X 0,Y 187.901,Z 410.93,A -85,B 0,C 180,E1 -24987.967,E2 -24987.967} C_VEL
LIN {X 0,Y 182.316,Z 396.825,A -85,B 0,C 180,E1 -24991.032,E2 -24991.032} C_VEL
LIN {X 0,Y 176.776,Z 384.263,A -85,B 0,C 180,E1 -24994.32,E2 -24994.32} C_VEL
LIN {X 0,Y 173.936,Z 379.086,A -85,B 0,C 180,E1 -24996.095,E2 -24996.095} C_VEL
LIN {X 0,Y 168.455,Z 370.471,A -85,B 0,C 180,E1 -24999.734,E2 -24999.734} C_VEL
LIN {X 0,Y 163.767,Z 363.55,A -85,B 0,C 180,E1 -25003.318,E2 -25003.318} C_VEL
LIN {X 0,Y 160.769,Z 359.24,A -85,B 0,C 180,E1 -25005.908,E2 -25005.908} C_VEL
LIN {X 0,Y 158.073,Z 355.399,A -85,B 0,C 180,E1 -25008.52,E2 -25008.52} C_VEL
LIN {X 0,Y 155.377,Z 351.821,A -85,B 0,C 180,E1 -25011.447,E2 -25011.447} C_VEL
LIN {X 0,Y 154.63,Z 350.563,A -85,B 0,C 180,E1 -25012.386,E2 -25012.386} C_VEL
LIN {X 0,Y 152.214,Z 347.731,A -85,B 0,C 180,E1 -25015.556,E2 -25015.556} C_VEL
LIN {X 0,Y 151.107,Z 345.693,A -85,B 0,C 180,E1 -25017.33,E2 -25017.33} C_VEL
LIN {X 0,Y 147.89,Z 342.082,A -85,B 0,C 180,E1 -25023.663,E2 -25023.663} C_VEL
LIN {X 0,Y 147.03,Z 340.245,A -85,B 0,C 180,E1 -25026.419,E2 -25026.419} C_VEL
LIN {X 0,Y 145.599,Z 339.902,A -85,B 0,C 180,E1 -25036.83,E2 -25036.83} C_VEL
LIN {X 0,Y 146.764,Z 340.559,A -85,B 0,C 180,E1 -25043.451,E2 -25043.451} C_VEL
LIN {X 0,Y 148.043,Z 343.632,A -85,B 0,C 180,E1 -25047.697,E2 -25047.697} C_VEL
LIN {X 0,Y 150.952,Z 346.204,A -85,B 0,C 180,E1 -25053.066,E2 -25053.066} C_VEL
LIN {X 0,Y 152.921,Z 349.471,A -85,B 0,C 180,E1 -25056.114,E2 -25056.114} C_VEL
LIN {X 0,Y 154.919,Z 351.378,A -85,B 0,C 180,E1 -25058.555,E2 -25058.555} C_VEL
LIN {X 0,Y 157.528,Z 355.116,A -85,B 0,C 180,E1 -25061.503,E2 -25061.503} C_VEL
LIN {X 0,Y 158.749,Z 356.598,A -85,B 0,C 180,E1 -25062.724,E2 -25062.724} C_VEL
LIN {X 0,Y 162.3,Z 361.529,A -85,B 0,C 180,E1 -25066.002,E2 -25066.002} C_VEL
LIN {X 0,Y 166.27,Z 367.243,A -85,B 0,C 180,E1 -25069.184,E2 -25069.184} C_VEL
LIN {X 0,Y 171.336,Z 374.935,A -85,B 0,C 180,E1 -25072.78,E2 -25072.78} C_VEL
LIN {X 0,Y 176.768,Z 383.919,A -85,B 0,C 180,E1 -25076.178,E2 -25076.178} C_VEL
LIN {X 0,Y 183.828,Z 396.59,A -85,B 0,C 180,E1 -25080.075,E2 -25080.075} C_VEL
LIN {X 0,Y 188.161,Z 405.342,A -85,B 0,C 180,E1 -25082.287,E2 -25082.287} C_VEL
LIN {X 0,Y 182.185,Z 470.236,A -85,B 0,C 180,E1 -25084.444,E2 -25084.444} C_VEL
LIN {X 0,Y 179.686,Z 485.956,A -85,B 0,C 180,E1 -25085.29,E2 -25085.29} C_VEL
LIN {X 0,Y 176.33,Z 501.287,A -85,B 0,C 180,E1 -25086.511,E2 -25086.511} C_VEL
LIN {X 0,Y 172.445,Z 515.039,A -85,B 0,C 180,E1 -25087.963,E2 -25087.963} C_VEL
LIN {X 0,Y 167.987,Z 528.317,A -85,B 0,C 180,E1 -25089.808,E2 -25089.808} C_VEL
LIN {X 0,Y 162.657,Z 541.722,A -85,B 0,C 180,E1 -25092.192,E2 -25092.192} C_VEL
LIN {X 0,Y 156.921,Z 554.295,A -85,B 0,C 180,E1 -25095.076,E2 -25095.076} C_VEL
LIN {X 0,Y 150.772,Z 566.373,A -85,B 0,C 180,E1 -25098.676,E2 -25098.676} C_VEL
LIN {X 0,Y 145.535,Z 576.022,A -85,B 0,C 180,E1 -25102.368,E2 -25102.368} C_VEL
LIN {X 0,Y 139.927,Z 585.69,A -85,B 0,C 180,E1 -25107.12,E2 -25107.12} C_VEL
LIN {X 0,Y 135.222,Z 593.678,A -85,B 0,C 180,E1 -25112.233,E2 -25112.233} C_VEL
LIN {X 0,Y 131.515,Z 600.203,A -85,B 0,C 180,E1 -25117.676,E2 -25117.676} C_VEL
LIN {X 0,Y 128.545,Z 606.104,A -85,B 0,C 180,E1 -25124.241,E2 -25124.241} C_VEL
LIN {X 0,Y 126.897,Z 609.683,A -85,B 0,C 180,E1 -25129.71,E2 -25129.71} C_VEL
LIN {X 0,Y 125.848,Z 612.872,A -85,B 0,C 180,E1 -25136.695,E2 -25136.695} C_VEL
LIN {X 0,Y 125.829,Z 614.541,A -85,B 0,C 180,E1 -25143.103,E2 -25143.103} C_VEL
LIN {X 0,Y 126.705,Z 615.11,A -85,B 0,C 180,E1 -25149.064,E2 -25149.064} C_VEL
LIN {X 0,Y 128.627,Z 614.616,A -85,B 0,C 180,E1 -25155.257,E2 -25155.257} C_VEL
LIN {X 0,Y 130.871,Z 613.525,A -85,B 0,C 180,E1 -25159.885,E2 -25159.885} C_VEL
LIN {X 0,Y 135.24,Z 610.84,A -85,B 0,C 180,E1 -25166.246,E2 -25166.246} C_VEL
LIN {X 0,Y 140.115,Z 607.408,A -85,B 0,C 180,E1 -25171.371,E2 -25171.371} C_VEL
LIN {X 0,Y 145.989,Z 602.898,A -85,B 0,C 180,E1 -25176.153,E2 -25176.153} C_VEL
LIN {X 0,Y 152.365,Z 597.616,A -85,B 0,C 180,E1 -25180.289,E2 -25180.289} C_VEL
LIN {X 0,Y 160.439,Z 590.256,A -85,B 0,C 180,E1 -25184.508,E2 -25184.508} C_VEL
LIN {X 0,Y 168.409,Z 582.187,A -85,B 0,C 180,E1 -25187.96,E2 -25187.96} C_VEL
LIN {X 0,Y 176.093,Z 573.462,A -85,B 0,C 180,E1 -25190.818,E2 -25190.818} C_VEL
LIN {X 0,Y 184.321,Z 563.001,A -85,B 0,C 180,E1 -25193.435,E2 -25193.435} C_VEL
LIN {X 0,Y 192.072,Z 551.677,A -85,B 0,C 180,E1 -25195.633,E2 -25195.633} C_VEL
LIN {X 0,Y 199.195,Z 539.728,A -85,B 0,C 180,E1 -25197.416,E2 -25197.416} C_VEL
LIN {X 0,Y 205.599,Z 527.148,A -85,B 0,C 180,E1 -25198.905,E2 -25198.905} C_VEL
LIN {X 0,Y 211.272,Z 513.821,A -85,B 0,C 180,E1 -25200.128,E2 -25200.128} C_VEL
LIN {X 0,Y 216.144,Z 499.678,A -85,B 0,C 180,E1 -25201.111,E2 -25201.111} C_VEL
LIN {X 0,Y 220.078,Z 484.837,A -85,B 0,C 180,E1 -25201.863,E2 -25201.863} C_VEL
LIN {X 0,Y 222.725,Z 471.085,A -85,B 0,C 180,E1 -25202.344,E2 -25202.344} C_VEL
LIN {X 0,Y 227.747,Z 429.163,A -85,B 0,C 180,E1 -25203.441,E2 -25203.441} C_VEL
LIN {X 0,Y 225.482,Z 423.105,A -85,B 0,C 180,E1 -25207.165,E2 -25207.165} C_VEL
LIN {X 0,Y 223.916,Z 419.515,A -85,B 0,C 180,E1 -25211.592,E2 -25211.592} C_VEL
LIN {X 0,Y 223.619,Z 419.382,A -85,B 0,C 180,E1 -25216.434,E2 -25216.434} C_VEL
LIN {X 0,Y 223.933,Z 419.87,A -85,B 0,C 180,E1 -25218.294,E2 -25218.294} C_VEL
LIN {X 0,Y 225.076,Z 423.14,A -85,B 0,C 180,E1 -25221.808,E2 -25221.808} C_VEL
LIN {X 0,Y 226.336,Z 427.43,A -85,B 0,C 180,E1 -25224.356,E2 -25224.356} C_VEL
LIN {X 0,Y 227.475,Z 431.895,A -85,B 0,C 180,E1 -25226.285,E2 -25226.285} C_VEL
LIN {X 0,Y 222.086,Z 476.279,A -85,B 0,C 180,E1 -25227.462,E2 -25227.462} C_VEL
LIN {X 0,Y 218.889,Z 491.692,A -85,B 0,C 180,E1 -25228.003,E2 -25228.003} C_VEL
LIN {X 0,Y 214.457,Z 506.991,A -85,B 0,C 180,E1 -25228.765,E2 -25228.765} C_VEL
LIN {X 0,Y 209.339,Z 520.809,A -85,B 0,C 180,E1 -25229.698,E2 -25229.698} C_VEL
LIN {X 0,Y 203.542,Z 533.602,A -85,B 0,C 180,E1 -25230.811,E2 -25230.811} C_VEL
LIN {X 0,Y 196.538,Z 546.733,A -85,B 0,C 180,E1 -25232.354,E2 -25232.354} C_VEL
LIN {X 0,Y 188.491,Z 559.624,A -85,B 0,C 180,E1 -25234.307,E2 -25234.307} C_VEL
LIN {X 0,Y 179.845,Z 571.65,A -85,B 0,C 180,E1 -25236.768,E2 -25236.768} C_VEL
LIN {X 0,Y 170.921,Z 582.482,A -85,B 0,C 180,E1 -25239.724,E2 -25239.724} C_VEL
LIN {X 0,Y 168.307,Z 584.963,A -85,B 0,C 180,E1 -25240.336,E2 -25240.336} C_VEL
LIN {X 0,Y 157.695,Z 592.629,A -85,B 0,C 180,E1 -25241.522,E2 -25241.522} C_VEL
LIN {X 0,Y 155.092,Z 594.745,A -85,B 0,C 180,E1 -25242.277,E2 -25242.277} C_VEL
LIN {X 0,Y 147.145,Z 601.839,A -85,B 0,C 180,E1 -25246.17,E2 -25246.17} C_VEL
LIN {X 0,Y 139.369,Z 608.211,A -85,B 0,C 180,E1 -25250.927,E2 -25250.927} C_VEL
LIN {X 0,Y 132.641,Z 613.255,A -85,B 0,C 180,E1 -25256.199,E2 -25256.199} C_VEL
LIN {X 0,Y 126.614,Z 617.416,A -85,B 0,C 180,E1 -25262.646,E2 -25262.646} C_VEL
LIN {X 0,Y 122.329,Z 620.215,A -85,B 0,C 180,E1 -25269.838,E2 -25269.838} C_VEL
LIN {X 0,Y 120.078,Z 621.516,A -85,B 0,C 180,E1 -25276.462,E2 -25276.462} C_VEL
LIN {X 0,Y 119.215,Z 621.67,A -85,B 0,C 180,E1 -25283.23,E2 -25283.23} C_VEL
LIN {X 0,Y 119.369,Z 620.698,A -85,B 0,C 180,E1 -25290.001,E2 -25290.001} C_VEL
LIN {X 0,Y 119.266,Z 618.496,A -85,B 0,C 180,E1 -25296.77,E2 -25296.77} C_VEL
LIN {X 0,Y 120.094,Z 615.021,A -85,B 0,C 180,E1 -25303.539,E2 -25303.539} C_VEL
LIN {X 0,Y 122.164,Z 610.18,A -85,B 0,C 180,E1 -25310.193,E2 -25310.193} C_VEL
LIN {X 0,Y 125.558,Z 603.835,A -85,B 0,C 180,E1 -25316.603,E2 -25316.603} C_VEL
LIN {X 0,Y 129.648,Z 596.944,A -85,B 0,C 180,E1 -25321.907,E2 -25321.907} C_VEL
LIN {X 0,Y 134.882,Z 588.598,A -85,B 0,C 180,E1 -25326.813,E2 -25326.813} C_VEL
LIN {X 0,Y 139.792,Z 580.014,A -85,B 0,C 180,E1 -25330.812,E2 -25330.812} C_VEL
LIN {X 0,Y 145.522,Z 569.969,A -85,B 0,C 180,E1 -25334.45,E2 -25334.45} C_VEL
LIN {X 0,Y 151.766,Z 558.006,A -85,B 0,C 180,E1 -25337.811,E2 -25337.811} C_VEL
LIN {X 0,Y 157.384,Z 546.105,A -85,B 0,C 180,E1 -25340.381,E2 -25340.381} C_VEL
LIN {X 0,Y 162.542,Z 533.6,A -85,B 0,C 180,E1 -25342.498,E2 -25342.498} C_VEL
LIN {X 0,Y 167.548,Z 519.272,A -85,B 0,C 180,E1 -25344.361,E2 -25344.361} C_VEL
LIN {X 0,Y 171.344,Z 506.288,A -85,B 0,C 180,E1 -25345.636,E2 -25345.636} C_VEL
LIN {X 0,Y 174.737,Z 491.54,A -85,B 0,C 180,E1 -25346.702,E2 -25346.702} C_VEL
LIN {X 0,Y 177.253,Z 475.987,A -85,B 0,C 180,E1 -25347.478,E2 -25347.478} C_VEL
LIN {X 0,Y 183.125,Z 413.306,A -85,B 0,C 180,E1 -25349.578,E2 -25349.578} C_VEL
LIN {X 0,Y 178.126,Z 400.479,A -85,B 0,C 180,E1 -25352.494,E2 -25352.494} C_VEL
LIN {X 0,Y 173.058,Z 388.544,A -85,B 0,C 180,E1 -25355.757,E2 -25355.757} C_VEL
LIN {X 0,Y 168.753,Z 381.084,A -85,B 0,C 180,E1 -25358.605,E2 -25358.605} C_VEL
LIN {X 0,Y 163.85,Z 373.37,A -85,B 0,C 180,E1 -25362.265,E2 -25362.265} C_VEL
LIN {X 0,Y 161.084,Z 369.252,A -85,B 0,C 180,E1 -25364.549,E2 -25364.549} C_VEL
LIN {X 0,Y 158.143,Z 364.858,A -85,B 0,C 180,E1 -25367.3,E2 -25367.3} C_VEL
LIN {X 0,Y 156.064,Z 361.779,A -85,B 0,C 180,E1 -25369.434,E2 -25369.434} C_VEL
LIN {X 0,Y 153.385,Z 357.962,A -85,B 0,C 180,E1 -25372.553,E2 -25372.553} C_VEL
LIN {X 0,Y 152.565,Z 356.844,A -85,B 0,C 180,E1 -25373.625,E2 -25373.625} C_VEL
LIN {X 0,Y 150.177,Z 353.515,A -85,B 0,C 180,E1 -25377.07,E2 -25377.07} C_VEL
LIN {X 0,Y 149.669,Z 352.47,A -85,B 0,C 180,E1 -25377.977,E2 -25377.977} C_VEL
LIN {X 0,Y 146.483,Z 348.566,A -85,B 0,C 180,E1 -25384.789,E2 -25384.789} C_VEL
LIN {X 0,Y 145.934,Z 347.325,A -85,B 0,C 180,E1 -25386.742,E2 -25386.742} C_VEL
LIN {X 0,Y 144.634,Z 346.911,A -85,B 0,C 180,E1 -25394.056,E2 -25394.056} C_VEL
LIN {X 0,Y 145.652,Z 347.492,A -85,B 0,C 180,E1 -25402.946,E2 -25402.946} C_VEL
LIN {X 0,Y 146.894,Z 350.586,A -85,B 0,C 180,E1 -25407.35,E2 -25407.35} C_VEL
LIN {X 0,Y 149.493,Z 353.008,A -85,B 0,C 180,E1 -25412.385,E2 -25412.385} C_VEL
LIN {X 0,Y 151.523,Z 356.307,A -85,B 0,C 180,E1 -25415.641,E2 -25415.641} C_VEL
LIN {X 0,Y 153.217,Z 358.066,A -85,B 0,C 180,E1 -25417.807,E2 -25417.807} C_VEL
LIN {X 0,Y 155.896,Z 361.865,A -85,B 0,C 180,E1 -25420.963,E2 -25420.963} C_VEL
LIN {X 0,Y 160.11,Z 367.813,A -85,B 0,C 180,E1 -25425.116,E2 -25425.116} C_VEL
LIN {X 0,Y 164.923,Z 374.897,A -85,B 0,C 180,E1 -25429.093,E2 -25429.093} C_VEL
LIN {X 0,Y 170.267,Z 383.637,A -85,B 0,C 180,E1 -25432.966,E2 -25432.966} C_VEL
LIN {X 0,Y 176.062,Z 393.829,A -85,B 0,C 180,E1 -25436.619,E2 -25436.619} C_VEL
LIN {X 0,Y 181.371,Z 404.02,A -85,B 0,C 180,E1 -25439.625,E2 -25439.625} C_VEL
LIN {X 0,Y 183.317,Z 407.976,A -85,B 0,C 180,E1 -25440.655,E2 -25440.655} C_VEL
LIN {X 0,Y 177.428,Z 470.51,A -85,B 0,C 180,E1 -25442.767,E2 -25442.767} C_VEL
LIN {X 0,Y 174.847,Z 486.24,A -85,B 0,C 180,E1 -25443.617,E2 -25443.617} C_VEL
LIN {X 0,Y 171.416,Z 501.427,A -85,B 0,C 180,E1 -25444.828,E2 -25444.828} C_VEL
LIN {X 0,Y 167.613,Z 514.507,A -85,B 0,C 180,E1 -25446.198,E2 -25446.198} C_VEL
LIN {X 0,Y 162.781,Z 528.468,A -85,B 0,C 180,E1 -25448.137,E2 -25448.137} C_VEL
LIN {X 0,Y 157.049,Z 542.354,A -85,B 0,C 180,E1 -25450.644,E2 -25450.644} C_VEL
LIN {X 0,Y 151.29,Z 554.465,A -85,B 0,C 180,E1 -25453.469,E2 -25453.469} C_VEL
LIN {X 0,Y 144.972,Z 566.412,A -85,B 0,C 180,E1 -25457.096,E2 -25457.096} C_VEL
LIN {X 0,Y 138.963,Z 576.934,A -85,B 0,C 180,E1 -25461.272,E2 -25461.272} C_VEL
LIN {X 0,Y 133.29,Z 586.218,A -85,B 0,C 180,E1 -25466.054,E2 -25466.054} C_VEL
LIN {X 0,Y 128.258,Z 594.361,A -85,B 0,C 180,E1 -25471.569,E2 -25471.569} C_VEL
LIN {X 0,Y 123.969,Z 601.597,A -85,B 0,C 180,E1 -25478.146,E2 -25478.146} C_VEL
LIN {X 0,Y 121.041,Z 607.199,A -85,B 0,C 180,E1 -25485.144,E2 -25485.144} C_VEL
LIN {X 0,Y 119.533,Z 610.462,A -85,B 0,C 180,E1 -25490.655,E2 -25490.655} C_VEL
LIN {X 0,Y 118.685,Z 613.197,A -85,B 0,C 180,E1 -25497.362,E2 -25497.362} C_VEL
LIN {X 0,Y 118.817,Z 614.794,A -85,B 0,C 180,E1 -25504.108,E2 -25504.108} C_VEL
LIN {X 0,Y 119.867,Z 615.317,A -85,B 0,C 180,E1 -25510.35,E2 -25510.35} C_VEL
LIN {X 0,Y 121.81,Z 614.892,A -85,B 0,C 180,E1 -25516.192,E2 -25516.192} C_VEL
LIN {X 0,Y 124.807,Z 613.573,A -85,B 0,C 180,E1 -25522.028,E2 -25522.028} C_VEL
LIN {X 0,Y 128.175,Z 611.728,A -85,B 0,C 180,E1 -25526.756,E2 -25526.756} C_VEL
LIN {X 0,Y 134.123,Z 607.975,A -85,B 0,C 180,E1 -25532.968,E2 -25532.968} C_VEL
LIN {X 0,Y 140.353,Z 603.588,A -85,B 0,C 180,E1 -25537.869,E2 -25537.869} C_VEL
LIN {X 0,Y 148.765,Z 597.013,A -85,B 0,C 180,E1 -25543.005,E2 -25543.005} C_VEL
LIN {X 0,Y 157.223,Z 589.654,A -85,B 0,C 180,E1 -25547.09,E2 -25547.09} C_VEL
LIN {X 0,Y 165.795,Z 581.273,A -85,B 0,C 180,E1 -25550.526,E2 -25550.526} C_VEL
LIN {X 0,Y 174.301,Z 571.914,A -85,B 0,C 180,E1 -25553.403,E2 -25553.403} C_VEL
LIN {X 0,Y 182.003,Z 562.331,A -85,B 0,C 180,E1 -25555.683,E2 -25555.683} C_VEL
LIN {X 0,Y 190.393,Z 550.38,A -85,B 0,C 180,E1 -25557.888,E2 -25557.888} C_VEL
LIN {X 0,Y 197.735,Z 538.192,A -85,B 0,C 180,E1 -25559.598,E2 -25559.598} C_VEL
LIN {X 0,Y 204.578,Z 524.749,A -85,B 0,C 180,E1 -25561.058,E2 -25561.058} C_VEL
LIN {X 0,Y 210.476,Z 510.602,A -85,B 0,C 180,E1 -25562.241,E2 -25562.241} C_VEL
LIN {X 0,Y 215.559,Z 495.247,A -85,B 0,C 180,E1 -25563.193,E2 -25563.193} C_VEL
LIN {X 0,Y 219.437,Z 479.428,A -85,B 0,C 180,E1 -25563.873,E2 -25563.873} C_VEL
LIN {X 0,Y 222.048,Z 462.988,A -85,B 0,C 180,E1 -25564.349,E2 -25564.349} C_VEL
LIN {X 0,Y 225.552,Z 433.913,A -85,B 0,C 180,E1 -25565.089,E2 -25565.089} C_VEL
LIN {X 0,Y 224.232,Z 429.878,A -85,B 0,C 180,E1 -25567.633,E2 -25567.633} C_VEL
LIN {X 0,Y 222.919,Z 426.547,A -85,B 0,C 180,E1 -25571.645,E2 -25571.645} C_VEL
LIN {X 0,Y 222.648,Z 426.406,A -85,B 0,C 180,E1 -25576.507,E2 -25576.507} C_VEL
LIN {X 0,Y 222.894,Z 426.883,A -85,B 0,C 180,E1 -25578.074,E2 -25578.074} C_VEL
LIN {X 0,Y 223.854,Z 430.01,A -85,B 0,C 180,E1 -25581.359,E2 -25581.359} C_VEL
LIN {X 0,Y 224.919,Z 434.031,A -85,B 0,C 180,E1 -25583.769,E2 -25583.769} C_VEL
LIN {X 0,Y 225.366,Z 436.081,A -85,B 0,C 180,E1 -25584.666,E2 -25584.666} C_VEL
LIN {X 0,Y 220.347,Z 475.669,A -85,B 0,C 180,E1 -25585.653,E2 -25585.653} C_VEL
LIN {X 0,Y 217.075,Z 491.192,A -85,B 0,C 180,E1 -25586.183,E2 -25586.183} C_VEL
LIN {X 0,Y 212.731,Z 505.999,A -85,B 0,C 180,E1 -25586.879,E2 -25586.879} C_VEL
LIN {X 0,Y 207.477,Z 519.989,A -85,B 0,C 180,E1 -25587.759,E2 -25587.759} C_VEL
LIN {X 0,Y 201.547,Z 532.849,A -85,B 0,C 180,E1 -25588.827,E2 -25588.827} C_VEL
LIN {X 0,Y 194.276,Z 546.198,A -85,B 0,C 180,E1 -25590.322,E2 -25590.322} C_VEL
LIN {X 0,Y 185.763,Z 559.382,A -85,B 0,C 180,E1 -25592.239,E2 -25592.239} C_VEL
LIN {X 0,Y 177.076,Z 571.04,A -85,B 0,C 180,E1 -25594.562,E2 -25594.562} C_VEL
LIN {X 0,Y 168.018,Z 581.707,A -85,B 0,C 180,E1 -25597.372,E2 -25597.372} C_VEL
LIN {X 0,Y 159.387,Z 590.636,A -85,B 0,C 180,E1 -25600.484,E2 -25600.484} C_VEL
LIN {X 0,Y 155.092,Z 594.745,A -85,B 0,C 180,E1 -25602.277,E2 -25602.277} C_VEL
LIN {X 0,Y 151.445,Z 597.795,A -85,B 0,C 180,E1 -25603.59,E2 -25603.59} C_VEL
LIN {X 0,Y 144.183,Z 602.487,A -85,B 0,C 180,E1 -25605.475,E2 -25605.475} C_VEL
LIN {X 0,Y 136.904,Z 606.709,A -85,B 0,C 180,E1 -25607.631,E2 -25607.631} C_VEL
LIN {X 0,Y 133.323,Z 608.926,A -85,B 0,C 180,E1 -25609.382,E2 -25609.382} C_VEL
LIN {X 0,Y 126.752,Z 613.422,A -85,B 0,C 180,E1 -25614.397,E2 -25614.397} C_VEL
LIN {X 0,Y 122.217,Z 616.332,A -85,B 0,C 180,E1 -25618.835,E2 -25618.835} C_VEL
LIN {X 0,Y 117.448,Z 619.146,A -85,B 0,C 180,E1 -25625.239,E2 -25625.239} C_VEL
LIN {X 0,Y 114.156,Z 620.871,A -85,B 0,C 180,E1 -25632.074,E2 -25632.074} C_VEL
LIN {X 0,Y 112.474,Z 621.533,A -85,B 0,C 180,E1 -25639.197,E2 -25639.197} C_VEL
LIN {X 0,Y 112.107,Z 621.043,A -85,B 0,C 180,E1 -25646.407,E2 -25646.407} C_VEL
LIN {X 0,Y 112.269,Z 620.364,A -85,B 0,C 180,E1 -25650.001,E2 -25650.001} C_VEL
LIN {X 0,Y 112.202,Z 618.057,A -85,B 0,C 180,E1 -25657.198,E2 -25657.198} C_VEL
LIN {X 0,Y 113.156,Z 614.474,A -85,B 0,C 180,E1 -25664.386,E2 -25664.386} C_VEL
LIN {X 0,Y 115.44,Z 609.515,A -85,B 0,C 180,E1 -25671.426,E2 -25671.426} C_VEL
LIN {X 0,Y 119.191,Z 603.05,A -85,B 0,C 180,E1 -25678.146,E2 -25678.146} C_VEL
LIN {X 0,Y 123.61,Z 596.037,A -85,B 0,C 180,E1 -25683.666,E2 -25683.666} C_VEL
LIN {X 0,Y 129.158,Z 587.567,A -85,B 0,C 180,E1 -25688.739,E2 -25688.739} C_VEL
LIN {X 0,Y 135.113,Z 577.777,A -85,B 0,C 180,E1 -25693.257,E2 -25693.257} C_VEL
LIN {X 0,Y 141.524,Z 566.773,A -85,B 0,C 180,E1 -25697.095,E2 -25697.095} C_VEL
LIN {X 0,Y 147.596,Z 555.336,A -85,B 0,C 180,E1 -25700.158,E2 -25700.158} C_VEL
LIN {X 0,Y 153.443,Z 542.911,A -85,B 0,C 180,E1 -25702.732,E2 -25702.732} C_VEL
LIN {X 0,Y 157.887,Z 532.281,A -85,B 0,C 180,E1 -25704.442,E2 -25704.442} C_VEL
LIN {X 0,Y 162.82,Z 518.54,A -85,B 0,C 180,E1 -25706.192,E2 -25706.192} C_VEL
LIN {X 0,Y 166.734,Z 505.404,A -85,B 0,C 180,E1 -25707.46,E2 -25707.46} C_VEL
LIN {X 0,Y 170.055,Z 491.285,A -85,B 0,C 180,E1 -25708.472,E2 -25708.472} C_VEL
LIN {X 0,Y 172.595,Z 476.054,A -85,B 0,C 180,E1 -25709.233,E2 -25709.233} C_VEL
LIN {X 0,Y 178.44,Z 415.685,A -85,B 0,C 180,E1 -25711.26,E2 -25711.26} C_VEL
LIN {X 0,Y 173.922,Z 403.807,A -85,B 0,C 180,E1 -25714.115,E2 -25714.115} C_VEL
LIN {X 0,Y 169.293,Z 392.651,A -85,B 0,C 180,E1 -25717.302,E2 -25717.302} C_VEL
LIN {X 0,Y 163.625,Z 382.923,A -85,B 0,C 180,E1 -25721.46,E2 -25721.46} C_VEL
LIN {X 0,Y 158.882,Z 375.482,A -85,B 0,C 180,E1 -25725.456,E2 -25725.456} C_VEL
LIN {X 0,Y 156.013,Z 371.088,A -85,B 0,C 180,E1 -25728.275,E2 -25728.275} C_VEL
LIN {X 0,Y 153.966,Z 368.005,A -85,B 0,C 180,E1 -25730.498,E2 -25730.498} C_VEL
LIN {X 0,Y 151.463,Z 364.113,A -85,B 0,C 180,E1 -25733.673,E2 -25733.673} C_VEL
LIN {X 0,Y 148.691,Z 360.22,A -85,B 0,C 180,E1 -25737.795,E2 -25737.795} C_VEL
LIN {X 0,Y 148.077,Z 359.134,A -85,B 0,C 180,E1 -25738.933,E2 -25738.933} C_VEL
LIN {X 0,Y 144.993,Z 354.659,A -85,B 0,C 180,E1 -25746.509,E2 -25746.509} C_VEL
LIN {X 0,Y 144.753,Z 354.209,A -85,B 0,C 180,E1 -25747.444,E2 -25747.444} C_VEL
LIN {X 0,Y 143.672,Z 353.978,A -85,B 0,C 180,E1 -25757.063,E2 -25757.063} C_VEL
LIN {X 0,Y 144.598,Z 354.607,A -85,B 0,C 180,E1 -25762.704,E2 -25762.704} C_VEL
LIN {X 0,Y 145.674,Z 357.424,A -85,B 0,C 180,E1 -25766.796,E2 -25766.796} C_VEL
LIN {X 0,Y 148.067,Z 359.808,A -85,B 0,C 180,E1 -25771.706,E2 -25771.706} C_VEL
LIN {X 0,Y 150.262,Z 363.339,A -85,B 0,C 180,E1 -25775.35,E2 -25775.35} C_VEL
LIN {X 0,Y 151.656,Z 364.89,A -85,B 0,C 180,E1 -25777.195,E2 -25777.195} C_VEL
LIN {X 0,Y 154.942,Z 369.706,A -85,B 0,C 180,E1 -25781.159,E2 -25781.159} C_VEL
LIN {X 0,Y 158.017,Z 374.195,A -85,B 0,C 180,E1 -25784.262,E2 -25784.262} C_VEL
LIN {X 0,Y 162.497,Z 381.099,A -85,B 0,C 180,E1 -25788.189,E2 -25788.189} C_VEL
LIN {X 0,Y 167.053,Z 388.769,A -85,B 0,C 180,E1 -25791.673,E2 -25791.673} C_VEL
LIN {X 0,Y 172.467,Z 398.5,A -85,B 0,C 180,E1 -25795.294,E2 -25795.294} C_VEL
LIN {X 0,Y 177.641,Z 408.733,A -85,B 0,C 180,E1 -25798.431,E2 -25798.431} C_VEL
LIN {X 0,Y 178.645,Z 410.856,A -85,B 0,C 180,E1 -25799.004,E2 -25799.004} C_VEL
LIN {X 0,Y 172.729,Z 470.966,A -85,B 0,C 180,E1 -25801.024,E2 -25801.024} C_VEL
LIN {X 0,Y 170.066,Z 486.656,A -85,B 0,C 180,E1 -25801.877,E2 -25801.877} C_VEL
LIN {X 0,Y 166.536,Z 501.729,A -85,B 0,C 180,E1 -25803.079,E2 -25803.079} C_VEL
LIN {X 0,Y 162.72,Z 514.454,A -85,B 0,C 180,E1 -25804.411,E2 -25804.411} C_VEL
LIN {X 0,Y 157.741,Z 528.449,A -85,B 0,C 180,E1 -25806.36,E2 -25806.36} C_VEL
LIN {X 0,Y 151.944,Z 542.019,A -85,B 0,C 180,E1 -25808.799,E2 -25808.799} C_VEL
LIN {X 0,Y 145.802,Z 554.525,A -85,B 0,C 180,E1 -25811.74,E2 -25811.74} C_VEL
LIN {X 0,Y 139.269,Z 566.376,A -85,B 0,C 180,E1 -25815.384,E2 -25815.384} C_VEL
LIN {X 0,Y 133.353,Z 576.312,A -85,B 0,C 180,E1 -25819.369,E2 -25819.369} C_VEL
LIN {X 0,Y 127.061,Z 586.188,A -85,B 0,C 180,E1 -25824.568,E2 -25824.568} C_VEL
LIN {X 0,Y 121.98,Z 594.002,A -85,B 0,C 180,E1 -25829.999,E2 -25829.999} C_VEL
LIN {X 0,Y 118.336,Z 599.664,A -85,B 0,C 180,E1 -25835.11,E2 -25835.11} C_VEL
LIN {X 0,Y 114.951,Z 605.521,A -85,B 0,C 180,E1 -25842.013,E2 -25842.013} C_VEL
LIN {X 0,Y 112.991,Z 609.371,A -85,B 0,C 180,E1 -25848.118,E2 -25848.118} C_VEL
LIN {X 0,Y 112.13,Z 611.307,A -85,B 0,C 180,E1 -25852.088,E2 -25852.088} C_VEL
LIN {X 0,Y 111.538,Z 613.516,A -85,B 0,C 180,E1 -25858.114,E2 -25858.114} C_VEL
LIN {X 0,Y 111.812,Z 615.045,A -85,B 0,C 180,E1 -25865.214,E2 -25865.214} C_VEL
LIN {X 0,Y 113.435,Z 615.492,A -85,B 0,C 180,E1 -25872.959,E2 -25872.959} C_VEL
LIN {X 0,Y 115.298,Z 615.093,A -85,B 0,C 180,E1 -25877.903,E2 -25877.903} C_VEL
LIN {X 0,Y 119.601,Z 613.33,A -85,B 0,C 180,E1 -25885.348,E2 -25885.348} C_VEL
LIN {X 0,Y 124.411,Z 610.801,A -85,B 0,C 180,E1 -25891.111,E2 -25891.111} C_VEL
LIN {X 0,Y 130.335,Z 607.278,A -85,B 0,C 180,E1 -25896.44,E2 -25896.44} C_VEL
LIN {X 0,Y 139.032,Z 601.378,A -85,B 0,C 180,E1 -25902.35,E2 -25902.35} C_VEL
LIN {X 0,Y 148.116,Z 594.407,A -85,B 0,C 180,E1 -25907.073,E2 -25907.073} C_VEL
LIN {X 0,Y 156.681,Z 587.018,A -85,B 0,C 180,E1 -25910.674,E2 -25910.674} C_VEL
LIN {X 0,Y 166.064,Z 577.843,A -85,B 0,C 180,E1 -25913.99,E2 -25913.99} C_VEL
LIN {X 0,Y 174.325,Z 568.66,A -85,B 0,C 180,E1 -25916.476,E2 -25916.476} C_VEL
LIN {X 0,Y 183.597,Z 556.878,A -85,B 0,C 180,E1 -25918.9,E2 -25918.9} C_VEL
LIN {X 0,Y 191.522,Z 545.109,A -85,B 0,C 180,E1 -25920.736,E2 -25920.736} C_VEL
LIN {X 0,Y 198.34,Z 533.353,A -85,B 0,C 180,E1 -25922.156,E2 -25922.156} C_VEL
LIN {X 0,Y 205.188,Z 519.289,A -85,B 0,C 180,E1 -25923.493,E2 -25923.493} C_VEL
LIN {X 0,Y 210.215,Z 506.679,A -85,B 0,C 180,E1 -25924.401,E2 -25924.401} C_VEL
LIN {X 0,Y 214.929,Z 491.759,A -85,B 0,C 180,E1 -25925.21,E2 -25925.21} C_VEL
LIN {X 0,Y 218.417,Z 476.751,A -85,B 0,C 180,E1 -25925.773,E2 -25925.773} C_VEL
LIN {X 0,Y 221.397,Z 456.256,A -85,B 0,C 180,E1 -25926.314,E2 -25926.314} C_VEL
LIN {X 0,Y 223.543,Z 438.715,A -85,B 0,C 180,E1 -25926.779,E2 -25926.779} C_VEL
LIN {X 0,Y 222.941,Z 436.524,A -85,B 0,C 180,E1 -25928.249,E2 -25928.249} C_VEL
